        CleaningLinesSolvent1and2();

        IF bMovementComplete THEN
            eRecoveryState    := E_RecoveryState.AgitateTime2;
            iStepCounter      := 0;
            bMovementComplete := FALSE;
        END_IF


    // ----------------------------------------------------------------------
    // AgitateTime2:
    //  - Second agitation time window after lines are cleaned.
    // ----------------------------------------------------------------------
    E_RecoveryState.AgitateTime2:

        AgitateTime2();

        IF bMovementComplete THEN
            eRecoveryState    := E_RecoveryState.Prime_Needles;
            iStepCounter      := 0;
            bMovementComplete := FALSE;
        END_IF


    // ----------------------------------------------------------------------
    // Prime_Needles:
    //  - Primes the needles and final tubing before filling vials.
    // ----------------------------------------------------------------------
    E_RecoveryState.Prime_Needles:

        PrimeNeedles();

        IF bMovementComplete THEN
            eRecoveryState    := E_RecoveryState.Fill_Vials_Row_1;
            iStepCounter      := 0;
            bMovementComplete := FALSE;
        END_IF


    // ----------------------------------------------------------------------
    // Fill_Vials_Row_1:
    //  - Fills the first row of vials.
    //  - Decides next state based on how many rows must be filled
    //    (iVialsToFill from recipe).
    // ----------------------------------------------------------------------
    E_RecoveryState.Fill_Vials_Row_1:

        Fill_Vials_Row_1();

        IF bMovementComplete THEN
            IF GVL_Recipe.stCurrentRecipe.stOtherParams.iVialsToFill > 1 THEN
                eRecoveryState := E_RecoveryState.Fill_Vials_Row_2;
            ELSE
                eRecoveryState := E_RecoveryState.Waste_Remaining_Solvent;
            END_IF

            bMovementComplete := FALSE;
            iStepCounter      := 0;
        END_IF


    // ----------------------------------------------------------------------
    // Fill_Vials_Row_2:
    //  - Fills the second row of vials (if required).
    // ----------------------------------------------------------------------
    E_RecoveryState.Fill_Vials_Row_2:

        Fill_Vials_Row_2();

        IF bMovementComplete THEN
            IF GVL_Recipe.stCurrentRecipe.stOtherParams.iVialsToFill > 2 THEN
                eRecoveryState := E_RecoveryState.Fill_Vials_Row_3;
            ELSE
                eRecoveryState := E_RecoveryState.Waste_Remaining_Solvent;
            END_IF

            bMovementComplete := FALSE;
            iStepCounter      := 0;
        END_IF


    // ----------------------------------------------------------------------
    // Fill_Vials_Row_3:
    //  - Fills the third row of vials (if required).
    // ----------------------------------------------------------------------
    E_RecoveryState.Fill_Vials_Row_3:

        Fill_Vials_Row_3();

        IF bMovementComplete THEN
            IF GVL_Recipe.stCurrentRecipe.stOtherParams.iVialsToFill > 3 THEN
                eRecoveryState := E_RecoveryState.Fill_Vials_Row_4;
            ELSE
                eRecoveryState := E_RecoveryState.Waste_Remaining_Solvent;
            END_IF

            bMovementComplete := FALSE;
            iStepCounter      := 0;
        END_IF


    // ----------------------------------------------------------------------
    // Fill_Vials_Row_4:
    //  - Fills the fourth row of vials (if required).
    // ----------------------------------------------------------------------
    E_RecoveryState.Fill_Vials_Row_4:

        Fill_Vials_Row_4();

        IF bMovementComplete THEN
            eRecoveryState    := E_RecoveryState.Waste_Remaining_Solvent;
            bMovementComplete := FALSE;
            iStepCounter      := 0;
        END_IF


    // ----------------------------------------------------------------------
    // Waste_Remaining_Solvent:
    //  - Directs any remaining solvent to waste containers.
    // ----------------------------------------------------------------------
    E_RecoveryState.Waste_Remaining_Solvent:

        WasteRemainingSolvent();

        IF bMovementComplete THEN
            eRecoveryState    := E_RecoveryState.Completed;
            bMovementComplete := FALSE;
            iStepCounter      := 0;
        END_IF


    // ----------------------------------------------------------------------
    // Completed:
    //  - Recovery phase has finished successfully.
    //  - Updates HMI and raises bSuccess.
    // ----------------------------------------------------------------------
    E_RecoveryState.Completed:

        GVL_HMI.HMIAnimation.sLoadTextRecovery   := 'Completed';
        GVL_HMI.HMIAnimation.rLoadBarRecovery    := 100.0;
        GVL_HMI.HMIAnimation.eIconStateRecovery  := E_IconState.Completed;

        bSuccess := TRUE;
        // bError stays FALSE here. If you later implement error transitions
        // to a dedicated Error state, set bError accordingly there.

END_CASE

ACTION AgitateTime1:
// ==========================================================================
// AgitateTime1
// --------------------------------------------------------------------------
// Purpose:
//   - Handles the first agitation timer window for the Recovery Phase.
//   - Uses tonAgitateTime1 and sets bMovementComplete when finished.
//
// Sequence (iStepCounter):
//   0) Check if Agitate Time 1 > 0. If zero, skip directly to step 3.
//   1) Start TON timer with recipe time tAgitate1Time.
//   2) Stop TON timer and move to completion.
//   3) Raise bMovementComplete to notify the caller state.
// ==========================================================================
CASE iStepCounter OF

    0:  // Check if Agitate Time 1 is greater than zero
        IF TIME_TO_DWORD(GVL_Recipe.stActiveRecipe.stOtherParams.tAgitate1Time / 1000) > 0 THEN
            // Update HMI text
            GVL_HMI.HMIAnimation.sLoadTextRecovery := 'Agitate Time 1';
            iStepCounter := 1;
        ELSE
            // No time configured → skip timer and mark as done
            iStepCounter := 3;
        END_IF

    1:  // Start Agitate Timer 1
        tonAgitateTime1(
            IN := TRUE,
            PT := GVL_Recipe.stActiveRecipe.stOtherParams.tAgitate1Time
        );

        // When timer finishes, proceed to stop it
        IF tonAgitateTime1.Q THEN
            iStepCounter := 2;
        END_IF

    2:  // Reset Agitate Timer 1
        tonAgitateTime1(
            IN := FALSE,
            PT := GVL_Recipe.stActiveRecipe.stOtherParams.tAgitate1Time
        );
        iStepCounter := 3;

    3:  // Signal completion to Recovery FSM
        bMovementComplete := TRUE;

END_CASE
END_ACTION

ACTION AgitateTime2:
// ==========================================================================
// AgitateTime2
// --------------------------------------------------------------------------
// Purpose:
//   - Handles the second agitation timer window for the Recovery Phase.
//   - Uses tonAgitateTime2 and sets bMovementComplete when finished.
//
// Sequence (iStepCounter):
//   0) Check if Agitate Time 2 > 0. If zero, skip directly to step 3.
//   1) Start TON timer with recipe time tAgitate2Time.
//   2) Stop TON timer and move to completion.
//   3) Raise bMovementComplete to notify the caller state.
// ==========================================================================
CASE iStepCounter OF

    0:  // Check if Agitate Time 2 is greater than zero
        IF TIME_TO_DWORD(GVL_Recipe.stActiveRecipe.stOtherParams.tAgitate2Time / 1000) > 0 THEN
            // Update HMI text
            GVL_HMI.HMIAnimation.sLoadTextRecovery := 'Agitate Time 2';
            iStepCounter := 1;
        ELSE
            // No time configured → skip timer and mark as done
            iStepCounter := 3;
        END_IF

    1:  // Start Agitate Timer 2
        tonAgitateTime2(
            IN := TRUE,
            PT := GVL_Recipe.stActiveRecipe.stOtherParams.tAgitate2Time
        );

        // When timer finishes, proceed to stop it
        IF tonAgitateTime2.Q THEN
            iStepCounter := 2;
        END_IF

    2:  // Reset Agitate Timer 2
        tonAgitateTime2(
            IN := FALSE,
            PT := GVL_Recipe.stActiveRecipe.stOtherParams.tAgitate2Time
        );
        iStepCounter := 3;

    3:  // Signal completion to Recovery FSM
        bMovementComplete := TRUE;

END_CASE
END_ACTION

ACTION CleaningLinesSolvent1:
// ==========================================================================
// CleaningLinesSolvent1
// --------------------------------------------------------------------------
// Purpose:
//   - Flush / clean the fluidic lines after using Solvent 1.
//   - Moves all valves to recirculation position (5).
//   - Pumps a larger volume through all paths to clean residual solvent.
//
// Sequence (iStepCounter):
//   0) Set HMI text and prepare.
//   1) Move all valves [1..5] to position 5 (Recirculation).
//   2) Calculate pump distances based on recipe volumes (Rinse 1) + dead volume.
//   3) Run all pumps [1..10] forward with higher velocity for cleaning.
//   4) Set bMovementComplete TRUE to notify FSM.
// ==========================================================================
CASE iStepCounter OF

    0:  // Initialize action / HMI
        GVL_HMI.HMIAnimation.sLoadTextRecovery := 'Cleaning Lines R1';
        iStepCounter := 1;

    1:  // Move valves [1..5] to position 5 (Recirculation)
        FOR i := 1 TO 5 DO
            IF NOT bMoveValveDone[i] THEN
                bMoveValveDone[i] := GVL_Motion.aValvesObj[i].MoveValve(
                    iPosition := 5,
                    rVelocity := GVL_Motion.aValves[i].rTargetVel,
                    rAcc      := GVL_Motion.aValves[i].rAcceleration,
                    rDec      := GVL_Motion.aValves[i].rDeceleration
                );
            END_IF
        END_FOR

        // Wait until all valves have completed their move
        IF bMoveValveDone[1] AND bMoveValveDone[2] AND bMoveValveDone[3]
           AND bMoveValveDone[4] AND bMoveValveDone[5]
        THEN
            // Reset valve flags and move to next step
            FOR i := 1 TO 5 DO
                bMoveValveDone[i] := FALSE;
            END_FOR
            iStepCounter := 2;
        END_IF

    2:  // Calculate pump distances for cleaning (based on Rinse 1 volume)
        // Factor 1.5 is used to add margin for extra cleaning volume
		(*
        fDistance[1]  := F_VolumeToSteps((GVL_Recipe.stActiveRecipe.stVolumes.aT_IC_Volume[1] +
                                          GVL_Motion.aPumps[1].Rotary.rDeadVolume) * 1.5, 1);
										  
        fDistance[2]  := F_VolumeToSteps((GVL_Recipe.stActiveRecipe.stVolumes.aS0_Volume[1] +
                                          GVL_Motion.aPumps[2].Rotary.rDeadVolume) * 1.5, 2);
										  
        fDistance[3]  := F_VolumeToSteps((GVL_Recipe.stActiveRecipe.stVolumes.aS1_Volume[1] +
                                          GVL_Motion.aPumps[3].Rotary.rDeadVolume) * 1.5, 3);
										  
        fDistance[4]  := F_VolumeToSteps((GVL_Recipe.stActiveRecipe.stVolumes.aS2_Volume[1] +
                                          GVL_Motion.aPumps[4].Rotary.rDeadVolume) * 1.5, 4);
										  
        fDistance[5]  := F_VolumeToSteps((GVL_Recipe.stActiveRecipe.stVolumes.aS3_Volume[1] +
                                          GVL_Motion.aPumps[5].Rotary.rDeadVolume) * 1.5, 5);
										  
        fDistance[6]  := F_VolumeToSteps((GVL_Recipe.stActiveRecipe.stVolumes.aS4_Volume[1] +
                                          GVL_Motion.aPumps[6].Rotary.rDeadVolume) * 1.5, 6);
										  
        fDistance[7]  := F_VolumeToSteps((GVL_Recipe.stActiveRecipe.stVolumes.aS5_Volume[1] +
                                          GVL_Motion.aPumps[7].Rotary.rDeadVolume) * 1.5, 7);
										  
        fDistance[8]  := F_VolumeToSteps((GVL_Recipe.stActiveRecipe.stVolumes.aS6_Volume[1] +
                                          GVL_Motion.aPumps[8].Rotary.rDeadVolume) * 1.5, 8);
										  
        fDistance[9]  := F_VolumeToSteps((GVL_Recipe.stActiveRecipe.stVolumes.aS7_Volume[1] +
                                          GVL_Motion.aPumps[9].Rotary.rDeadVolume) * 1.5, 9);
										  
        fDistance[10] := F_VolumeToSteps((GVL_Recipe.stActiveRecipe.stVolumes.aF_Volume[1] +
                                          GVL_Motion.aPumps[10].Rotary.rDeadVolume) * 1.5, 10);
		*)
		
		// Constant volume for cleaning lines. change#15/01/26
		FOR i := 1 TO 10 DO
			fDistance[i]  := F_VolumeToSteps( 100 + GVL_Motion.aPumps[i].Rotary.rDeadVolume, i);
		END_FOR
		
        iStepCounter := 3;

    3:  // Start rotary pumps with calculated distances [positive movement]
        FOR i := 1 TO 10 DO
            IF NOT bMovePumpDone[i] THEN
                bMovePumpDone[i] := GVL_Motion.aPumpsRotary[i].MoveRelative(
                    Distance := fDistance[i],
                    Velocity := GVL_Settings.stPumpParameters.iRunVelocity * 6,
                    Acc      := GVL_Settings.stPumpParameters.iRunVelocity * 3,
                    Dec      := GVL_Settings.stPumpParameters.iRunVelocity * 3
                );
            END_IF
        END_FOR

        // Wait until every pump has completed the move
        IF bMovePumpDone[1] AND bMovePumpDone[2] AND bMovePumpDone[3] AND bMovePumpDone[4] AND
           bMovePumpDone[5] AND bMovePumpDone[6] AND bMovePumpDone[7] AND bMovePumpDone[8] AND
           bMovePumpDone[9] AND bMovePumpDone[10]
        THEN
            FOR i := 1 TO 10 DO
                bMovePumpDone[i] := FALSE;
            END_FOR
            iStepCounter := 4;
        END_IF

    4:  // Signal completion to Recovery FSM
        bMovementComplete := TRUE;

END_CASE
END_ACTION

ACTION CleaningLinesSolvent1and2:
// ==========================================================================
// CleaningLinesSolvent1and2
// --------------------------------------------------------------------------
// Purpose:
//   - Flush / clean all lines that carried Solvent 1 and Solvent 2.
//   - Uses the combined volumes of both rinses to determine a larger
//     cleaning volume per pump.
//
// Sequence (iStepCounter):
//   0) Set HMI text.
//   1) Move all valves [1..5] to position 5 (Recirculation).
//   2) Calculate pump distances from sum of Rinse 1 + Rinse 2 volumes.
//   3) Run all pumps [1..10] forward with higher velocity.
//   4) Set bMovementComplete TRUE.
// ==========================================================================
CASE iStepCounter OF

    0:  // Initialize action / HMI
        GVL_HMI.HMIAnimation.sLoadTextRecovery := 'Cleaning Lines';
        iStepCounter := 1;

    1:  // Move valves [1..5] to position 5 (Recirculation)
        FOR i := 1 TO 5 DO
            IF NOT bMoveValveDone[i] THEN
                bMoveValveDone[i] := GVL_Motion.aValvesObj[i].MoveValve(
                    iPosition := 5,
                    rVelocity := GVL_Motion.aValves[i].rTargetVel,
                    rAcc      := GVL_Motion.aValves[i].rAcceleration,
                    rDec      := GVL_Motion.aValves[i].rDeceleration
                );
            END_IF
        END_FOR

        IF bMoveValveDone[1] AND bMoveValveDone[2] AND bMoveValveDone[3]
           AND bMoveValveDone[4] AND bMoveValveDone[5]
        THEN
            FOR i := 1 TO 5 DO
                bMoveValveDone[i] := FALSE;
            END_FOR
            iStepCounter := 2;
        END_IF

    2:  // Calculate distances using combined volumes (Rinse 1 + Rinse 2)
        fDistance[1]  := F_VolumeToSteps((GVL_Recipe.stActiveRecipe.stVolumes.aT_IC_Volume[1] +
                                          GVL_Recipe.stActiveRecipe.stVolumes.aT_IC_Volume[2] +
                                          GVL_Motion.aPumps[1].Rotary.rDeadVolume) * 1.5, 1);
										  
        fDistance[2]  := F_VolumeToSteps((GVL_Recipe.stActiveRecipe.stVolumes.aS0_Volume[1] +
                                          GVL_Recipe.stActiveRecipe.stVolumes.aS0_Volume[2] +
                                          GVL_Motion.aPumps[2].Rotary.rDeadVolume) * 1.5, 2);
										  
        fDistance[3]  := F_VolumeToSteps((GVL_Recipe.stActiveRecipe.stVolumes.aS1_Volume[1] +
                                          GVL_Recipe.stActiveRecipe.stVolumes.aS1_Volume[2] +
                                          GVL_Motion.aPumps[3].Rotary.rDeadVolume) * 1.5, 3);
										  
        fDistance[4]  := F_VolumeToSteps((GVL_Recipe.stActiveRecipe.stVolumes.aS2_Volume[1] +
                                          GVL_Recipe.stActiveRecipe.stVolumes.aS2_Volume[2] +
                                          GVL_Motion.aPumps[4].Rotary.rDeadVolume) * 1.5, 4);
										  
        fDistance[5]  := F_VolumeToSteps((GVL_Recipe.stActiveRecipe.stVolumes.aS3_Volume[1] +
                                          GVL_Recipe.stActiveRecipe.stVolumes.aS3_Volume[2] +
                                          GVL_Motion.aPumps[5].Rotary.rDeadVolume) * 1.5, 5);
										  
        fDistance[6]  := F_VolumeToSteps((GVL_Recipe.stActiveRecipe.stVolumes.aS4_Volume[1] +
                                          GVL_Recipe.stActiveRecipe.stVolumes.aS4_Volume[2] +
                                          GVL_Motion.aPumps[6].Rotary.rDeadVolume) * 1.5, 6);
										  
        fDistance[7]  := F_VolumeToSteps((GVL_Recipe.stActiveRecipe.stVolumes.aS5_Volume[1] +
                                          GVL_Recipe.stActiveRecipe.stVolumes.aS5_Volume[2] +
                                          GVL_Motion.aPumps[7].Rotary.rDeadVolume) * 1.5, 7);
										  
        fDistance[8]  := F_VolumeToSteps((GVL_Recipe.stActiveRecipe.stVolumes.aS6_Volume[1] +
                                          GVL_Recipe.stActiveRecipe.stVolumes.aS6_Volume[2] +
                                          GVL_Motion.aPumps[8].Rotary.rDeadVolume) * 1.5, 8);
										  
        fDistance[9]  := F_VolumeToSteps((GVL_Recipe.stActiveRecipe.stVolumes.aS7_Volume[1] +
                                          GVL_Recipe.stActiveRecipe.stVolumes.aS7_Volume[2] +
                                          GVL_Motion.aPumps[9].Rotary.rDeadVolume) * 1.5, 9);
										  
        fDistance[10] := F_VolumeToSteps((GVL_Recipe.stActiveRecipe.stVolumes.aF_Volume[1] +
                                          GVL_Recipe.stActiveRecipe.stVolumes.aF_Volume[2] +
                                          GVL_Motion.aPumps[10].Rotary.rDeadVolume) * 1.5, 10);

        iStepCounter := 3;

    3:  // Run pumps with calculated distances [positive movement]
        FOR i := 1 TO 10 DO
            IF NOT bMovePumpDone[i] THEN
                bMovePumpDone[i] := GVL_Motion.aPumpsRotary[i].MoveRelative(
                    Distance := fDistance[i],
                    Velocity := GVL_Settings.stPumpParameters.iRunVelocity * 6,
                    Acc      := GVL_Settings.stPumpParameters.iRunVelocity * 3,
                    Dec      := GVL_Settings.stPumpParameters.iRunVelocity * 3
                );
            END_IF
        END_FOR

        IF bMovePumpDone[1] AND bMovePumpDone[2] AND bMovePumpDone[3] AND bMovePumpDone[4] AND
           bMovePumpDone[5] AND bMovePumpDone[6] AND bMovePumpDone[7] AND bMovePumpDone[8] AND
           bMovePumpDone[9] AND bMovePumpDone[10]
        THEN
            FOR i := 1 TO 10 DO
                bMovePumpDone[i] := FALSE;
            END_FOR
            iStepCounter := 4;
        END_IF

    4:  // Signal completion to Recovery FSM
        bMovementComplete := TRUE;

END_CASE
END_ACTION

METHOD PRIVATE EstimateTotalTime : REAL
VAR_INPUT
END_VAR
VAR
	i : INT;
	iRow : INT;
    rTotalTime : LREAL := 0.0;
    rMaxPumpTime : REAL;
    rTmpTime : REAL;
	aPumpVolume : ARRAY[1..10] OF REAL;
END_VAR
// --- MOTORS M2 and M3 ---
// Movements are sequential, so times are summed
rTotalTime := rTotalTime
    + (ABS(GVL_Settings.stMachineParam.aM2Position[3] - GVL_Settings.stMachineParam.aM2Position[1]) / GVL_Settings.stMachineParam.rM2Velocity) * 4
    + (ABS(GVL_Settings.stMachineParam.aM3Position[4] - GVL_Settings.stMachineParam.aM3Position[1]) / GVL_Settings.stMachineParam.rM3Velocity) * 4;

// --- VALVES ---
// Valves move in parallel, so estimate per group of 5 valves per switch
// Estimated 0.8s per position change, 8 total changes
rTotalTime := rTotalTime + 0.8 * 8;


// --- TIMERS ---
// Add the Agitation and Soak durations directly (in seconds)
rTotalTime := rTotalTime + TO_REAL(GVL_Recipe.stActiveRecipe.stOtherParams.tAgitate1Time) / 1000.0;
rTotalTime := rTotalTime + TO_REAL(GVL_Recipe.stActiveRecipe.stOtherParams.tAgitate2Time) / 1000.0;
rTotalTime := rTotalTime + TO_REAL(GVL_Recipe.stActiveRecipe.stOtherParams.tSoakTime) / 1000.0;


// --- PUMPS ---
// Pumps move in parallel. We always use the slowest pump as reference for each phase.

// Metering Solvent 1
rMaxPumpTime := 0;
aPumpVolume[1] := GVL_Recipe.stActiveRecipe.stVolumes.aT_IC_Volume[1] + 10;
aPumpVolume[2] := GVL_Recipe.stActiveRecipe.stVolumes.aS0_Volume[1] + 10;
aPumpVolume[3] := GVL_Recipe.stActiveRecipe.stVolumes.aS1_Volume[1] + 10;
aPumpVolume[4] := GVL_Recipe.stActiveRecipe.stVolumes.aS2_Volume[1] + 10;
aPumpVolume[5] := GVL_Recipe.stActiveRecipe.stVolumes.aS3_Volume[1] + 10;
aPumpVolume[6] := GVL_Recipe.stActiveRecipe.stVolumes.aS4_Volume[1] + 10;
aPumpVolume[7] := GVL_Recipe.stActiveRecipe.stVolumes.aS5_Volume[1] + 10;
aPumpVolume[8] := GVL_Recipe.stActiveRecipe.stVolumes.aS6_Volume[1] + 10;
aPumpVolume[9] := GVL_Recipe.stActiveRecipe.stVolumes.aS7_Volume[1] + 10;
aPumpVolume[10] := GVL_Recipe.stActiveRecipe.stVolumes.aF_Volume[1] + 10;

FOR i := 1 TO 10 DO
    rTmpTime := F_VolumeToSteps(rVolume := aPumpVolume[i], iPumpIndex := i) / GVL_Motion.aPumps[i].Rotary.rSpeed;
    IF rTmpTime > rMaxPumpTime THEN rMaxPumpTime := rTmpTime; END_IF
END_FOR
rTotalTime := rTotalTime + rMaxPumpTime;

// Metering Solvent 2
rMaxPumpTime := 0;
aPumpVolume[1] := GVL_Recipe.stActiveRecipe.stVolumes.aT_IC_Volume[2] + 10;
aPumpVolume[2] := GVL_Recipe.stActiveRecipe.stVolumes.aS0_Volume[2] + 10;
aPumpVolume[3] := GVL_Recipe.stActiveRecipe.stVolumes.aS1_Volume[2] + 10;
aPumpVolume[4] := GVL_Recipe.stActiveRecipe.stVolumes.aS2_Volume[2] + 10;
aPumpVolume[5] := GVL_Recipe.stActiveRecipe.stVolumes.aS3_Volume[2] + 10;
aPumpVolume[6] := GVL_Recipe.stActiveRecipe.stVolumes.aS4_Volume[2] + 10;
aPumpVolume[7] := GVL_Recipe.stActiveRecipe.stVolumes.aS5_Volume[2] + 10;
aPumpVolume[8] := GVL_Recipe.stActiveRecipe.stVolumes.aS6_Volume[2] + 10;
aPumpVolume[9] := GVL_Recipe.stActiveRecipe.stVolumes.aS7_Volume[2] + 10;
aPumpVolume[10] := GVL_Recipe.stActiveRecipe.stVolumes.aF_Volume[2] + 10;
FOR i := 1 TO 10 DO
    rTmpTime := F_VolumeToSteps(rVolume := aPumpVolume[i], iPumpIndex := i) / GVL_Motion.aPumps[i].Rotary.rSpeed;
    IF rTmpTime > rMaxPumpTime THEN rMaxPumpTime := rTmpTime; END_IF
END_FOR
rTotalTime := rTotalTime + rMaxPumpTime;

// Prime Needles
rMaxPumpTime := 0;
FOR i := 1 TO 10 DO
    rTmpTime := F_VolumeToSteps(rVolume := GVL_Recipe.stActiveRecipe.stOtherParams.rVialPrimeVol + 20, iPumpIndex := i) / GVL_Motion.aPumps[i].Rotary.rSpeed;
    IF rTmpTime > rMaxPumpTime THEN rMaxPumpTime := rTmpTime; END_IF
END_FOR
rTotalTime := rTotalTime + rMaxPumpTime;

// Fill Vials Rows 1–4
FOR iRow := 1 TO GVL_Recipe.stActiveRecipe.stOtherParams.iVialsToFill DO
    rMaxPumpTime := 0;
    FOR i := 1 TO 10 DO
        IF iRow = 1 THEN
            rTmpTime := F_VolumeToSteps(rVolume := GVL_Recipe.stActiveRecipe.stOtherParams.rVial1FillVol, iPumpIndex := i) / GVL_Motion.aPumps[i].Rotary.rSpeed;
        ELSE
            rTmpTime := F_VolumeToSteps(rVolume := GVL_Recipe.stActiveRecipe.stOtherParams.rVials2_4FillVol, iPumpIndex := i) / GVL_Motion.aPumps[i].Rotary.rSpeed;
        END_IF
        IF rTmpTime > rMaxPumpTime THEN 
			rMaxPumpTime := rTmpTime; 
		END_IF
    END_FOR
    rTotalTime := rTotalTime + rMaxPumpTime;
END_FOR

// Waste Remaining Solvent
rMaxPumpTime := 0;

FOR i := 1 TO 10 DO
    rTmpTime := F_VolumeToSteps(rVolume := GVL_Recipe.stActiveRecipe.stVolumes.aT_IC_Volume[1] + GVL_Recipe.stActiveRecipe.stVolumes.aT_IC_Volume[2], iPumpIndex := i) / GVL_Motion.aPumps[i].Rotary.rSpeed;
    IF rTmpTime > rMaxPumpTime THEN
 		rMaxPumpTime := rTmpTime; 
	END_IF
	
END_FOR
rTotalTime := rTotalTime + rMaxPumpTime;

EstimateTotalTime := rTotalTime + 180;
END_METHOD

ACTION Fill_Vials_Row_1:
// ==========================================================================
// Fill_Vials_Row_1
// --------------------------------------------------------------------------
// Purpose:
//   - Fill the first row of vials using the Recovery Phase solvent mixture.
//   - Move M3 (horizontal) to vial row 1 position and M2 (vertical) down to
//     the vial level.
//   - Pump the volume configured as rVial1FillVol into each vial.
//
// Sequence (iStepCounter):
//   0) Initialize HMI text and move to step 1.
//   1) Set all valves [1..5] to position 6 (Needles).
//   2) Move M3 to vial row 1 (horizontal) and M2 down to vial height.
//   3) Compute pump distances based on rVial1FillVol.
//   4) Run pumps [1..10] backward (negative Distance) to dispense volume.
//   5) Move M2 back to home (vertical).
//   6) Set bMovementComplete := TRUE to notify the Recovery FSM.
// ==========================================================================
CASE iStepCounter OF

    0: // Initialize HMI info for Row 1 filling
        GVL_HMI.HMIAnimation.sLoadTextRecovery := 'Fill Vials R1';
        // Optionally: GVL_HMI.HMIAnimation.rLoadBarRecovery := 70;
        iStepCounter := 1;

    1: // Set valves [1..5] to position 6 (Needles)
        FOR i := 1 TO 5 DO
            IF NOT bMoveValveDone[i] THEN
                bMoveValveDone[i] := GVL_Motion.aValvesObj[i].MoveValve(
                    iPosition := 6,
                    rVelocity := GVL_Motion.aValves[i].rTargetVel,
                    rAcc      := GVL_Motion.aValves[i].rAcceleration,
                    rDec      := GVL_Motion.aValves[i].rDeceleration
                );
            END_IF
        END_FOR

        // Wait for all valves to finish the movement
        IF bMoveValveDone[1] AND bMoveValveDone[2] AND bMoveValveDone[3]
           AND bMoveValveDone[4] AND bMoveValveDone[5]
        THEN
            // Reset valve flags and go to next step
            FOR i := 1 TO 5 DO
                bMoveValveDone[i] := FALSE;
            END_FOR
            iStepCounter := 2;
        END_IF

    2: // M2 and M3 motors movement to vial row 1 position
        // Step 2.1: Move M3 (horizontal) to Row 1 (AboveVialSet1)
        IF NOT bMoveM3 THEN
            bMoveM3 := GVL_Motion.aMotors[3].MoveAbsolute(
                rPosition := GVL_Settings.stMachineParam.aM3Position[2], // Vial row 1
                rVelocity := GVL_Settings.stMachineParam.rM3Velocity,
                rAcc      := GVL_Settings.stMachineParam.rM3Accleration,
                rDec      := GVL_Settings.stMachineParam.rM3Deceleration
            );
        END_IF

        // Step 2.2: After M3 is at row 1, move M2 (vertical) down to vial height
        IF NOT bMoveM2 AND bMoveM3 THEN
            bMoveM2 := GVL_Motion.aMotors[2].MoveAbsolute(
                rPosition := GVL_Settings.stMachineParam.aM2Position[3], // Fill position
                rVelocity := GVL_Settings.stMachineParam.rM2Velocity,
                rAcc      := GVL_Settings.stMachineParam.rM2Accleration,
                rDec      := GVL_Settings.stMachineParam.rM2Deceleration
            );
        END_IF

        // When both motors reach their positions, clear flags and go to step 3
        IF bMoveM2 AND bMoveM3 THEN
            bMoveM2      := FALSE;
            bMoveM3      := FALSE;
            iStepCounter := 3;
        END_IF

    3: // Calculate distance (steps) for each pump based on rVial1FillVol
        fDistance[1]  := F_VolumeToSteps(
            rVolume    := GVL_Recipe.stActiveRecipe.stOtherParams.rVial1FillVol,
            iPumpIndex := 1
        );
        fDistance[2]  := F_VolumeToSteps(
            rVolume    := GVL_Recipe.stActiveRecipe.stOtherParams.rVial1FillVol,
            iPumpIndex := 2
        );
        fDistance[3]  := F_VolumeToSteps(
            rVolume    := GVL_Recipe.stActiveRecipe.stOtherParams.rVial1FillVol,
            iPumpIndex := 3
        );
        fDistance[4]  := F_VolumeToSteps(
            rVolume    := GVL_Recipe.stActiveRecipe.stOtherParams.rVial1FillVol,
            iPumpIndex := 4
        );
        fDistance[5]  := F_VolumeToSteps(
            rVolume    := GVL_Recipe.stActiveRecipe.stOtherParams.rVial1FillVol,
            iPumpIndex := 5
        );
        fDistance[6]  := F_VolumeToSteps(
            rVolume    := GVL_Recipe.stActiveRecipe.stOtherParams.rVial1FillVol,
            iPumpIndex := 6
        );
        fDistance[7]  := F_VolumeToSteps(
            rVolume    := GVL_Recipe.stActiveRecipe.stOtherParams.rVial1FillVol,
            iPumpIndex := 7
        );
        fDistance[8]  := F_VolumeToSteps(
            rVolume    := GVL_Recipe.stActiveRecipe.stOtherParams.rVial1FillVol,
            iPumpIndex := 8
        );
        fDistance[9]  := F_VolumeToSteps(
            rVolume    := GVL_Recipe.stActiveRecipe.stOtherParams.rVial1FillVol,
            iPumpIndex := 9
        );
        fDistance[10] := F_VolumeToSteps(
            rVolume    := GVL_Recipe.stActiveRecipe.stOtherParams.rVial1FillVol,
            iPumpIndex := 10
        );

        iStepCounter := 4;

    4: // Pump by distance (deg/s → steps) [negative movement = dispensing to vials]
        FOR i := 1 TO 10 DO
            IF NOT bMovePumpDone[i] THEN
                bMovePumpDone[i] := GVL_Motion.aPumpsRotary[i].MoveRelative(
                    Distance := -fDistance[i],   // negative → pushing out to vials
                    Velocity := GVL_Settings.stPumpParameters.iMeterVelocity * 6,
                    Acc      := GVL_Settings.stPumpParameters.iMeterVelocity * 3,
                    Dec      := GVL_Settings.stPumpParameters.iMeterVelocity * 3
                );
            END_IF
        END_FOR

        // Wait until all pumps finish their moves
        IF bMovePumpDone[1]  AND bMovePumpDone[2]  AND bMovePumpDone[3]  AND
           bMovePumpDone[4]  AND bMovePumpDone[5]  AND bMovePumpDone[6]  AND
           bMovePumpDone[7]  AND bMovePumpDone[8]  AND bMovePumpDone[9]  AND
           bMovePumpDone[10]
        THEN
            FOR i := 1 TO 10 DO
                bMovePumpDone[i] := FALSE;
            END_FOR
            iStepCounter := 5;
        END_IF

    5: // Move M2 (vertical) back to home position
        IF NOT bMoveM2 THEN
            bMoveM2 := GVL_Motion.aMotors[2].MoveAbsolute(
                rPosition := GVL_Settings.stMachineParam.aM2Position[1], // home
                rVelocity := GVL_Settings.stMachineParam.rM2Velocity,
                rAcc      := GVL_Settings.stMachineParam.rM2Accleration,
                rDec      := GVL_Settings.stMachineParam.rM2Deceleration
            );
        END_IF

        // When M2 is home, clear flag and go to final step
        IF bMoveM2 THEN
            bMoveM2      := FALSE;
            iStepCounter := 6;
        END_IF

    6: // Notify Recovery FSM that Row 1 filling is completed
        bMovementComplete := TRUE;

END_CASE
END_ACTION

ACTION Fill_Vials_Row_2:
// ==========================================================================
// Fill_Vials_Row_2
// --------------------------------------------------------------------------
// Purpose:
//   - Fill the second row of vials using the same volume used for rows 2–4.
//   - Move M3 (horizontal) to vial row 2 and M2 (vertical) down to vial level.
//   - Pump the volume configured as rVials2_4FillVol into each vial.
//
// Sequence (iStepCounter):
//   0) Initialize HMI text and move to step 1.
//   1) Set all valves [1..5] to position 6 (Needles).
//   2) Move M3 to vial row 2 (AboveVialSet1 + VialSetSpacing) and M2 down.
//   3) Compute pump distances based on rVials2_4FillVol.
//   4) Run pumps [1..10] backward to dispense volume.
//   5) Move M2 back to home (vertical).
//   6) Set bMovementComplete := TRUE.
// ==========================================================================
CASE iStepCounter OF

    0: // Initialize HMI info for Row 2 filling
        GVL_HMI.HMIAnimation.sLoadTextRecovery := 'Fill Vials R2';
        // Optionally: GVL_HMI.HMIAnimation.rLoadBarRecovery := 75;
        iStepCounter := 1;

    1: // Set valves [1..5] to position 6 (Needles)
        FOR i := 1 TO 5 DO
            IF NOT bMoveValveDone[i] THEN
                bMoveValveDone[i] := GVL_Motion.aValvesObj[i].MoveValve(
                    iPosition := 6,
                    rVelocity := GVL_Motion.aValves[i].rTargetVel,
                    rAcc      := GVL_Motion.aValves[i].rAcceleration,
                    rDec      := GVL_Motion.aValves[i].rDeceleration
                );
            END_IF
        END_FOR

        IF bMoveValveDone[1] AND bMoveValveDone[2] AND bMoveValveDone[3]
           AND bMoveValveDone[4] AND bMoveValveDone[5]
        THEN
            FOR i := 1 TO 5 DO
                bMoveValveDone[i] := FALSE;
            END_FOR
            iStepCounter := 2;
        END_IF

    2: // M2 and M3 movement to vial row 2
        // Step 2.1: M3 → row 2 = AboveVialSet1 + 1 * VialSetSpacing
        IF NOT bMoveM3 THEN
            bMoveM3 := GVL_Motion.aMotors[3].MoveAbsolute(
                rPosition := GVL_Settings.stMachineParam.aM3Position[2] +
                             (1 * GVL_Settings.stMachineParam.aM3Position[3]),
                // comment: AboveVialSet1 + (1 * VialSetSpacing)
                rVelocity := GVL_Settings.stMachineParam.rM3Velocity,
                rAcc      := GVL_Settings.stMachineParam.rM3Accleration,
                rDec      := GVL_Settings.stMachineParam.rM3Deceleration
            );
        END_IF

        // Step 2.2: after M3 movement, bring M2 down to fill position
        IF NOT bMoveM2 AND bMoveM3 THEN
            bMoveM2 := GVL_Motion.aMotors[2].MoveAbsolute(
                rPosition := GVL_Settings.stMachineParam.aM2Position[3], // Fill position
                rVelocity := GVL_Settings.stMachineParam.rM2Velocity,
                rAcc      := GVL_Settings.stMachineParam.rM2Accleration,
                rDec      := GVL_Settings.stMachineParam.rM2Deceleration
            );
        END_IF

        IF bMoveM2 AND bMoveM3 THEN
            bMoveM2      := FALSE;
            bMoveM3      := FALSE;
            iStepCounter := 3;
        END_IF

    3: // Calculate distances for each pump based on rVials2_4FillVol
        fDistance[1]  := F_VolumeToSteps(
            rVolume    := GVL_Recipe.stActiveRecipe.stOtherParams.rVials2_4FillVol,
            iPumpIndex := 1
        );
        fDistance[2]  := F_VolumeToSteps(
            rVolume    := GVL_Recipe.stActiveRecipe.stOtherParams.rVials2_4FillVol,
            iPumpIndex := 2
        );
        fDistance[3]  := F_VolumeToSteps(
            rVolume    := GVL_Recipe.stActiveRecipe.stOtherParams.rVials2_4FillVol,
            iPumpIndex := 3
        );
        fDistance[4]  := F_VolumeToSteps(
            rVolume    := GVL_Recipe.stActiveRecipe.stOtherParams.rVials2_4FillVol,
            iPumpIndex := 4
        );
        fDistance[5]  := F_VolumeToSteps(
            rVolume    := GVL_Recipe.stActiveRecipe.stOtherParams.rVials2_4FillVol,
            iPumpIndex := 5
        );
        fDistance[6]  := F_VolumeToSteps(
            rVolume    := GVL_Recipe.stActiveRecipe.stOtherParams.rVials2_4FillVol,
            iPumpIndex := 6
        );
        fDistance[7]  := F_VolumeToSteps(
            rVolume    := GVL_Recipe.stActiveRecipe.stOtherParams.rVials2_4FillVol,
            iPumpIndex := 7
        );
        fDistance[8]  := F_VolumeToSteps(
            rVolume    := GVL_Recipe.stActiveRecipe.stOtherParams.rVials2_4FillVol,
            iPumpIndex := 8
        );
        fDistance[9]  := F_VolumeToSteps(
            rVolume    := GVL_Recipe.stActiveRecipe.stOtherParams.rVials2_4FillVol,
            iPumpIndex := 9
        );
        fDistance[10] := F_VolumeToSteps(
            rVolume    := GVL_Recipe.stActiveRecipe.stOtherParams.rVials2_4FillVol,
            iPumpIndex := 10
        );

        iStepCounter := 4;

    4: // Pump by distance (negative movement = dispensing to vials)
        FOR i := 1 TO 10 DO
            IF NOT bMovePumpDone[i] THEN
                bMovePumpDone[i] := GVL_Motion.aPumpsRotary[i].MoveRelative(
                    Distance := -fDistance[i],
                    Velocity := GVL_Settings.stPumpParameters.iMeterVelocity * 6,
                    Acc      := GVL_Settings.stPumpParameters.iMeterVelocity * 3,
                    Dec      := GVL_Settings.stPumpParameters.iMeterVelocity * 3
                );
            END_IF
        END_FOR

        IF bMovePumpDone[1]  AND bMovePumpDone[2]  AND bMovePumpDone[3]  AND
           bMovePumpDone[4]  AND bMovePumpDone[5]  AND bMovePumpDone[6]  AND
           bMovePumpDone[7]  AND bMovePumpDone[8]  AND bMovePumpDone[9]  AND
           bMovePumpDone[10]
        THEN
            FOR i := 1 TO 10 DO
                bMovePumpDone[i] := FALSE;
            END_FOR
            iStepCounter := 5;
        END_IF

    5: // Move M2 back to home position
        IF NOT bMoveM2 THEN
            bMoveM2 := GVL_Motion.aMotors[2].MoveAbsolute(
                rPosition := GVL_Settings.stMachineParam.aM2Position[1], // home
                rVelocity := GVL_Settings.stMachineParam.rM2Velocity,
                rAcc      := GVL_Settings.stMachineParam.rM2Accleration,
                rDec      := GVL_Settings.stMachineParam.rM2Deceleration
            );
        END_IF

        IF bMoveM2 THEN
            bMoveM2      := FALSE;
            iStepCounter := 6;
        END_IF

    6: // Notify Recovery FSM that Row 2 filling is completed
        bMovementComplete := TRUE;

END_CASE
END_ACTION

ACTION Fill_Vials_Row_3:
// ==========================================================================
// Fill_Vials_Row_3
// --------------------------------------------------------------------------
// Purpose:
//   - Fill the third row of vials using rVials2_4FillVol.
//   - Move M3 (horizontal) to row 3 and M2 (vertical) down to vials.
//   - Pump the configured volume into each vial.
//
// Sequence (iStepCounter):
//   0) Initialize HMI text.
//   1) Set valves [1..5] to position 6 (Needles).
//   2) Move M3 to vial row 3 (AboveVialSet1 + 2 * VialSetSpacing) and M2 down.
//   3) Compute pump distances based on rVials2_4FillVol.
//   4) Pump backward to dispense.
//   5) Move M2 back to home.
//   6) bMovementComplete := TRUE.
// ==========================================================================
CASE iStepCounter OF

    0: // Initialize HMI info for Row 3 filling
        GVL_HMI.HMIAnimation.sLoadTextRecovery := 'Fill Vials R3';
        iStepCounter := 1;

    1: // Set valves [1..5] to position 6 (Needles)
        FOR i := 1 TO 5 DO
            IF NOT bMoveValveDone[i] THEN
                bMoveValveDone[i] := GVL_Motion.aValvesObj[i].MoveValve(
                    iPosition := 6,
                    rVelocity := GVL_Motion.aValves[i].rTargetVel,
                    rAcc      := GVL_Motion.aValves[i].rAcceleration,
                    rDec      := GVL_Motion.aValves[i].rDeceleration
                );
            END_IF
        END_FOR

        IF bMoveValveDone[1] AND bMoveValveDone[2] AND bMoveValveDone[3]
           AND bMoveValveDone[4] AND bMoveValveDone[5]
        THEN
            FOR i := 1 TO 5 DO
                bMoveValveDone[i] := FALSE;
            END_FOR
            iStepCounter := 2;
        END_IF

    2: // M2 and M3 movement to vial row 3
        // Step 2.1: M3 → row 3 = AboveVialSet1 + 2 * VialSetSpacing
        IF NOT bMoveM3 THEN
            bMoveM3 := GVL_Motion.aMotors[3].MoveAbsolute(
                rPosition := GVL_Settings.stMachineParam.aM3Position[2] +
                             (2 * GVL_Settings.stMachineParam.aM3Position[3]),
                // comment: AboveVialSet1 + (2 * VialSetSpacing)
                rVelocity := GVL_Settings.stMachineParam.rM3Velocity,
                rAcc      := GVL_Settings.stMachineParam.rM3Accleration,
                rDec      := GVL_Settings.stMachineParam.rM3Deceleration
            );
        END_IF

        // Step 2.2: after M3 movement, bring M2 down to fill position
        IF NOT bMoveM2 AND bMoveM3 THEN
            bMoveM2 := GVL_Motion.aMotors[2].MoveAbsolute(
                rPosition := GVL_Settings.stMachineParam.aM2Position[3], // Fill position
                rVelocity := GVL_Settings.stMachineParam.rM2Velocity,
                rAcc      := GVL_Settings.stMachineParam.rM2Accleration,
                rDec      := GVL_Settings.stMachineParam.rM2Deceleration
            );
        END_IF

        IF bMoveM2 AND bMoveM3 THEN
            bMoveM2      := FALSE;
            bMoveM3      := FALSE;
            iStepCounter := 3;
        END_IF

    3: // Calculate distances for each pump based on rVials2_4FillVol
        fDistance[1]  := F_VolumeToSteps(
            rVolume    := GVL_Recipe.stActiveRecipe.stOtherParams.rVials2_4FillVol,
            iPumpIndex := 1
        );
        fDistance[2]  := F_VolumeToSteps(
            rVolume    := GVL_Recipe.stActiveRecipe.stOtherParams.rVials2_4FillVol,
            iPumpIndex := 2
        );
        fDistance[3]  := F_VolumeToSteps(
            rVolume    := GVL_Recipe.stActiveRecipe.stOtherParams.rVials2_4FillVol,
            iPumpIndex := 3
        );
        fDistance[4]  := F_VolumeToSteps(
            rVolume    := GVL_Recipe.stActiveRecipe.stOtherParams.rVials2_4FillVol,
            iPumpIndex := 4
        );
        fDistance[5]  := F_VolumeToSteps(
            rVolume    := GVL_Recipe.stActiveRecipe.stOtherParams.rVials2_4FillVol,
            iPumpIndex := 5
        );
        fDistance[6]  := F_VolumeToSteps(
            rVolume    := GVL_Recipe.stActiveRecipe.stOtherParams.rVials2_4FillVol,
            iPumpIndex := 6
        );
        fDistance[7]  := F_VolumeToSteps(
            rVolume    := GVL_Recipe.stActiveRecipe.stOtherParams.rVials2_4FillVol,
            iPumpIndex := 7
        );
        fDistance[8]  := F_VolumeToSteps(
            rVolume    := GVL_Recipe.stActiveRecipe.stOtherParams.rVials2_4FillVol,
            iPumpIndex := 8
        );
        fDistance[9]  := F_VolumeToSteps(
            rVolume    := GVL_Recipe.stActiveRecipe.stOtherParams.rVials2_4FillVol,
            iPumpIndex := 9
        );
        fDistance[10] := F_VolumeToSteps(
            rVolume    := GVL_Recipe.stActiveRecipe.stOtherParams.rVials2_4FillVol,
            iPumpIndex := 10
        );

        iStepCounter := 4;

    4: // Pump by distance (negative movement = dispensing to vials)
        FOR i := 1 TO 10 DO
            IF NOT bMovePumpDone[i] THEN
                bMovePumpDone[i] := GVL_Motion.aPumpsRotary[i].MoveRelative(
                    Distance := -fDistance[i],
                    Velocity := GVL_Settings.stPumpParameters.iMeterVelocity * 6,
                    Acc      := GVL_Settings.stPumpParameters.iMeterVelocity * 3,
                    Dec      := GVL_Settings.stPumpParameters.iMeterVelocity * 3
                );
            END_IF
        END_FOR

        IF bMovePumpDone[1]  AND bMovePumpDone[2]  AND bMovePumpDone[3]  AND
           bMovePumpDone[4]  AND bMovePumpDone[5]  AND bMovePumpDone[6]  AND
           bMovePumpDone[7]  AND bMovePumpDone[8]  AND bMovePumpDone[9]  AND
           bMovePumpDone[10]
        THEN
            FOR i := 1 TO 10 DO
                bMovePumpDone[i] := FALSE;
            END_FOR
            iStepCounter := 5;
        END_IF

    5: // Move M2 back to home position
        IF NOT bMoveM2 THEN
            bMoveM2 := GVL_Motion.aMotors[2].MoveAbsolute(
                rPosition := GVL_Settings.stMachineParam.aM2Position[1],
                rVelocity := GVL_Settings.stMachineParam.rM2Velocity,
                rAcc      := GVL_Settings.stMachineParam.rM2Accleration,
                rDec      := GVL_Settings.stMachineParam.rM2Deceleration
            );
        END_IF

        IF bMoveM2 THEN
            bMoveM2      := FALSE;
            iStepCounter := 6;
        END_IF

    6: // Notify Recovery FSM that Row 3 filling is completed
        bMovementComplete := TRUE;

END_CASE
END_ACTION

ACTION Fill_Vials_Row_4:
// ==========================================================================
// Fill_Vials_Row_4
// --------------------------------------------------------------------------
// Purpose:
//   - Fill the fourth row of vials using rVials2_4FillVol.
//   - Move M3 (horizontal) to row 4 and M2 (vertical) down to vials.
//   - Pump the configured volume into each vial.
//
// Sequence (iStepCounter):
//   0) Initialize HMI text.
//   1) Set valves [1..5] to position 6 (Needles).
//   2) Move M3 to vial row 4 (AboveVialSet1 + 3 * VialSetSpacing) and M2 down.
//   3) Compute pump distances based on rVials2_4FillVol.
//   4) Pump backward to dispense.
//   5) Move M2 back to home.
//   6) bMovementComplete := TRUE.
// ==========================================================================
CASE iStepCounter OF

    0: // Initialize HMI info for Row 4 filling
        GVL_HMI.HMIAnimation.sLoadTextRecovery := 'Fill Vials R4';
        iStepCounter := 1;

    1: // Set valves [1..5] to position 6 (Needles)
        FOR i := 1 TO 5 DO
            IF NOT bMoveValveDone[i] THEN
                bMoveValveDone[i] := GVL_Motion.aValvesObj[i].MoveValve(
                    iPosition := 6,
                    rVelocity := GVL_Motion.aValves[i].rTargetVel,
                    rAcc      := GVL_Motion.aValves[i].rAcceleration,
                    rDec      := GVL_Motion.aValves[i].rDeceleration
                );
            END_IF
        END_FOR

        IF bMoveValveDone[1] AND bMoveValveDone[2] AND bMoveValveDone[3]
           AND bMoveValveDone[4] AND bMoveValveDone[5]
        THEN
            FOR i := 1 TO 5 DO
                bMoveValveDone[i] := FALSE;
            END_FOR
            iStepCounter := 2;
        END_IF

    2: // M2 and M3 movement to vial row 4
        // Step 2.1: M3 → row 4 = AboveVialSet1 + 3 * VialSetSpacing
        IF NOT bMoveM3 THEN
            bMoveM3 := GVL_Motion.aMotors[3].MoveAbsolute(
                rPosition := GVL_Settings.stMachineParam.aM3Position[2] +
                             (3 * GVL_Settings.stMachineParam.aM3Position[3]),
                // comment: AboveVialSet1 + (3 * VialSetSpacing)
                rVelocity := GVL_Settings.stMachineParam.rM3Velocity,
                rAcc      := GVL_Settings.stMachineParam.rM3Accleration,
                rDec      := GVL_Settings.stMachineParam.rM3Deceleration
            );
        END_IF

        // Step 2.2: M2 down to fill position after M3 movement
        IF NOT bMoveM2 AND bMoveM3 THEN
            bMoveM2 := GVL_Motion.aMotors[2].MoveAbsolute(
                rPosition := GVL_Settings.stMachineParam.aM2Position[3], // Fill position
                rVelocity := GVL_Settings.stMachineParam.rM2Velocity,
                rAcc      := GVL_Settings.stMachineParam.rM2Accleration,
                rDec      := GVL_Settings.stMachineParam.rM2Deceleration
            );
        END_IF

        IF bMoveM2 AND bMoveM3 THEN
            bMoveM2      := FALSE;
            bMoveM3      := FALSE;
            iStepCounter := 3;
        END_IF

    3: // Calculate distances for each pump based on rVials2_4FillVol
        fDistance[1]  := F_VolumeToSteps(
            rVolume    := GVL_Recipe.stActiveRecipe.stOtherParams.rVials2_4FillVol,
            iPumpIndex := 1
        );
        fDistance[2]  := F_VolumeToSteps(
            rVolume    := GVL_Recipe.stActiveRecipe.stOtherParams.rVials2_4FillVol,
            iPumpIndex := 2
        );
        fDistance[3]  := F_VolumeToSteps(
            rVolume    := GVL_Recipe.stActiveRecipe.stOtherParams.rVials2_4FillVol,
            iPumpIndex := 3
        );
        fDistance[4]  := F_VolumeToSteps(
            rVolume    := GVL_Recipe.stActiveRecipe.stOtherParams.rVials2_4FillVol,
            iPumpIndex := 4
        );
        fDistance[5]  := F_VolumeToSteps(
            rVolume    := GVL_Recipe.stActiveRecipe.stOtherParams.rVials2_4FillVol,
            iPumpIndex := 5
        );
        fDistance[6]  := F_VolumeToSteps(
            rVolume    := GVL_Recipe.stActiveRecipe.stOtherParams.rVials2_4FillVol,
            iPumpIndex := 6
        );
        fDistance[7]  := F_VolumeToSteps(
            rVolume    := GVL_Recipe.stActiveRecipe.stOtherParams.rVials2_4FillVol,
            iPumpIndex := 7
        );
        fDistance[8]  := F_VolumeToSteps(
            rVolume    := GVL_Recipe.stActiveRecipe.stOtherParams.rVials2_4FillVol,
            iPumpIndex := 8
        );
        fDistance[9]  := F_VolumeToSteps(
            rVolume    := GVL_Recipe.stActiveRecipe.stOtherParams.rVials2_4FillVol,
            iPumpIndex := 9
        );
        fDistance[10] := F_VolumeToSteps(
            rVolume    := GVL_Recipe.stActiveRecipe.stOtherParams.rVials2_4FillVol,
            iPumpIndex := 10
        );

        iStepCounter := 4;

    4: // Pump by distance (negative movement = dispensing to vials)
        FOR i := 1 TO 10 DO
            IF NOT bMovePumpDone[i] THEN
                bMovePumpDone[i] := GVL_Motion.aPumpsRotary[i].MoveRelative(
                    Distance := -fDistance[i],
                    Velocity := GVL_Settings.stPumpParameters.iMeterVelocity * 6,
                    Acc      := GVL_Settings.stPumpParameters.iMeterVelocity * 3,
                    Dec      := GVL_Settings.stPumpParameters.iMeterVelocity * 3
                );
            END_IF
        END_FOR

        IF bMovePumpDone[1]  AND bMovePumpDone[2]  AND bMovePumpDone[3]  AND
           bMovePumpDone[4]  AND bMovePumpDone[5]  AND bMovePumpDone[6]  AND
           bMovePumpDone[7]  AND bMovePumpDone[8]  AND bMovePumpDone[9]  AND
           bMovePumpDone[10]
        THEN
            FOR i := 1 TO 10 DO
                bMovePumpDone[i] := FALSE;
            END_FOR
            iStepCounter := 5;
        END_IF

    5: // Move M2 back to home position
        IF NOT bMoveM2 THEN
            bMoveM2 := GVL_Motion.aMotors[2].MoveAbsolute(
                rPosition := GVL_Settings.stMachineParam.aM2Position[1],
                rVelocity := GVL_Settings.stMachineParam.rM2Velocity,
                rAcc      := GVL_Settings.stMachineParam.rM2Accleration,
                rDec      := GVL_Settings.stMachineParam.rM2Deceleration
            );
        END_IF

        IF bMoveM2 THEN
            bMoveM2      := FALSE;
            iStepCounter := 6;
        END_IF

    6: // Notify Recovery FSM that Row 4 filling is completed
        bMovementComplete := TRUE;

END_CASE
END_ACTION

METHOD PRIVATE GetPumpVolume : REAL
VAR_INPUT
	iPump : INT;  // Pump number 1..10
    iStep : INT;  // 1..4 [step Rinse 1 | Rinse 2 | Wash 1 | Wash 2] 
END_VAR
VAR
    volume : REAL;
END_VAR
CASE iPump OF
    1: volume := GVL_Recipe.stVolumes.aT_IC_Volume[iStep];
    2: volume := GVL_Recipe.stVolumes.aS0_Volume[iStep];
    3: volume := GVL_Recipe.stVolumes.aS1_Volume[iStep];
    4: volume := GVL_Recipe.stVolumes.aS2_Volume[iStep];
    5: volume := GVL_Recipe.stVolumes.aS3_Volume[iStep];
    6: volume := GVL_Recipe.stVolumes.aS4_Volume[iStep];
    7: volume := GVL_Recipe.stVolumes.aS5_Volume[iStep];
    8: volume := GVL_Recipe.stVolumes.aS6_Volume[iStep];
    9: volume := GVL_Recipe.stVolumes.aS7_Volume[iStep];
    10: volume := GVL_Recipe.stVolumes.aF_Volume[iStep];
    ELSE
        volume := 0.0;
END_CASE

GetPumpVolume := volume;
END_METHOD

ACTION MeteringSolvent1:
// ==========================================================================
// MeteringSolvent1
// --------------------------------------------------------------------------
// Purpose:
//   - Meter Solvent 1 volumes from each Andersen stage into the fluidic path.
//   - Positions valves according to recipe aSolventN[1].
//   - Moves all 10 pumps by a distance equivalent to the configured volumes.
//
// Sequence (iStepCounter):
//   0) Set HMI text.
//   1) Ensure solenoids are in IDLE position (via gSetSolenoidControl.Idle()).
//   2) Move all valves [1..5] to solvent-1 position (recipe-dependent).
//   3) Calculate pump distances for metering (Rinse 1 + dead volume).
//   4) Run all pumps forward at metering velocity.
//   5) Set bMovementComplete TRUE.
// ==========================================================================
CASE iStepCounter OF

    0:  // Initialize action / HMI
        GVL_HMI.HMIAnimation.sLoadTextRecovery := 'Metering Rinse 1';
        iStepCounter := 1;

    1:  // Initialization: wait solenoids at IDLE (safety/flow configuration)
        // fbSolenoidControl could also be used if re-enabled in the future
        // fbSolenoidControl(bExecute := TRUE, eSolenoidSet := E_SolenoidSet.IDLE);

        IF GVL_IO.gSetSolenoidControl.Idle() THEN
            iStepCounter := 2;
        END_IF

    2:  // Set valves for Rinse 1 (position comes from aSolventN[1])
        FOR i := 1 TO 5 DO
            IF NOT bMoveValveDone[i] THEN
                bMoveValveDone[i] := GVL_Motion.aValvesObj[i].MoveValve(
                    iPosition := GVL_Recipe.stActiveRecipe.stSolventsTimes.aSolventN[1],
                    rVelocity := GVL_Motion.aValves[i].rTargetVel,
                    rAcc      := GVL_Motion.aValves[i].rAcceleration,
                    rDec      := GVL_Motion.aValves[i].rDeceleration
                );
            END_IF
        END_FOR

        IF bMoveValveDone[1] AND bMoveValveDone[2] AND bMoveValveDone[3]
           AND bMoveValveDone[4] AND bMoveValveDone[5]
        THEN
            FOR i := 1 TO 5 DO
                bMoveValveDone[i] := FALSE;
            END_FOR
            iStepCounter := 3;
        END_IF

    3:  // Calculate the distance for each pump (Rinse 1 + dead volume)
        fDistance[1]  := F_VolumeToSteps(GVL_Recipe.stActiveRecipe.stVolumes.aT_IC_Volume[1] +
                                         GVL_Motion.aPumps[1].Rotary.rDeadVolume, 1);
										 
        fDistance[2]  := F_VolumeToSteps(GVL_Recipe.stActiveRecipe.stVolumes.aS0_Volume[1] +
                                         GVL_Motion.aPumps[2].Rotary.rDeadVolume, 2);
										 
        fDistance[3]  := F_VolumeToSteps(GVL_Recipe.stActiveRecipe.stVolumes.aS1_Volume[1] +
                                         GVL_Motion.aPumps[3].Rotary.rDeadVolume, 3);
										 
        fDistance[4]  := F_VolumeToSteps(GVL_Recipe.stActiveRecipe.stVolumes.aS2_Volume[1] +
                                         GVL_Motion.aPumps[4].Rotary.rDeadVolume, 4);
										 
        fDistance[5]  := F_VolumeToSteps(GVL_Recipe.stActiveRecipe.stVolumes.aS3_Volume[1] +
                                         GVL_Motion.aPumps[5].Rotary.rDeadVolume, 5);
										 
        fDistance[6]  := F_VolumeToSteps(GVL_Recipe.stActiveRecipe.stVolumes.aS4_Volume[1] +
                                         GVL_Motion.aPumps[6].Rotary.rDeadVolume, 6);
										 
        fDistance[7]  := F_VolumeToSteps(GVL_Recipe.stActiveRecipe.stVolumes.aS5_Volume[1] +
                                         GVL_Motion.aPumps[7].Rotary.rDeadVolume, 7);
										 
        fDistance[8]  := F_VolumeToSteps(GVL_Recipe.stActiveRecipe.stVolumes.aS6_Volume[1] +
                                         GVL_Motion.aPumps[8].Rotary.rDeadVolume, 8);
										 
        fDistance[9]  := F_VolumeToSteps(GVL_Recipe.stActiveRecipe.stVolumes.aS7_Volume[1] +
                                         GVL_Motion.aPumps[9].Rotary.rDeadVolume, 9);
										 
        fDistance[10] := F_VolumeToSteps(GVL_Recipe.stActiveRecipe.stVolumes.aF_Volume[1] +
                                         GVL_Motion.aPumps[10].Rotary.rDeadVolume, 10);

        iStepCounter := 4;

    4:  // Perform rotary movement for metering (positive movement)
        FOR i := 1 TO 10 DO
            IF NOT bMovePumpDone[i] THEN
                bMovePumpDone[i] := GVL_Motion.aPumpsRotary[i].MoveRelative(
                    Distance := fDistance[i],
                    Velocity := GVL_Settings.stPumpParameters.iMeterVelocity * 6,
                    Acc      := GVL_Settings.stPumpParameters.iMeterVelocity * 6,
                    Dec      := GVL_Settings.stPumpParameters.iMeterVelocity
                );
            END_IF
        END_FOR

        IF bMovePumpDone[1] AND bMovePumpDone[2] AND bMovePumpDone[3] AND bMovePumpDone[4] AND
           bMovePumpDone[5] AND bMovePumpDone[6] AND bMovePumpDone[7] AND bMovePumpDone[8] AND
           bMovePumpDone[9] AND bMovePumpDone[10]
        THEN
            FOR i := 1 TO 10 DO
                bMovePumpDone[i] := FALSE;
            END_FOR
            iStepCounter := 5;
        END_IF

    5:  // Signal completion to Recovery FSM
        bMovementComplete := TRUE;

END_CASE
END_ACTION

ACTION MeteringSolvent2:
// ==========================================================================
// MeteringSolvent2
// --------------------------------------------------------------------------
// Purpose:
//   - Meter Solvent 2 volumes from each Andersen stage into the fluidic path.
//   - Positions valves according to recipe aSolventN[2].
//   - Moves all 10 pumps by distance equivalent to Rinse 2 volumes.
//
// Sequence (iStepCounter):
//   0) Set HMI text.
//   1) Ensure solenoids are in IDLE position.
//   2) Move valves [1..5] to solvent-2 position (recipe-dependent).
//   3) Calculate pump distances (Rinse 2 + dead volume).
//   4) Run all pumps forward at metering velocity.
//   5) Set bMovementComplete TRUE.
// ==========================================================================
CASE iStepCounter OF

    0:  // Initialize action / HMI
        GVL_HMI.HMIAnimation.sLoadTextRecovery := 'Metering Rinse 2';
        iStepCounter := 1;

    1:  // Initialization: wait solenoids at IDLE
        // fbSolenoidControl(bExecute := TRUE, eSolenoidSet := E_SolenoidSet.IDLE);

        IF GVL_IO.gSetSolenoidControl.Idle() THEN
            iStepCounter := 2;
        END_IF

    2:  // Set valves for Rinse 2 (position comes from aSolventN[2])
        FOR i := 1 TO 5 DO
            IF NOT bMoveValveDone[i] THEN
                bMoveValveDone[i] := GVL_Motion.aValvesObj[i].MoveValve(
                    iPosition := GVL_Recipe.stActiveRecipe.stSolventsTimes.aSolventN[2],
                    rVelocity := GVL_Motion.aValves[i].rTargetVel,
                    rAcc      := GVL_Motion.aValves[i].rAcceleration,
                    rDec      := GVL_Motion.aValves[i].rDeceleration
                );
            END_IF
        END_FOR

        IF bMoveValveDone[1] AND bMoveValveDone[2] AND bMoveValveDone[3]
           AND bMoveValveDone[4] AND bMoveValveDone[5]
        THEN
            FOR i := 1 TO 5 DO
                bMoveValveDone[i] := FALSE;
            END_FOR
            iStepCounter := 3;
        END_IF

    3:  // Calculate the distance for each pump (Rinse 2 + dead volume)
        fDistance[1]  := F_VolumeToSteps(GVL_Recipe.stActiveRecipe.stVolumes.aT_IC_Volume[2] +
                                         GVL_Motion.aPumps[1].Rotary.rDeadVolume, 1);
										 
        fDistance[2]  := F_VolumeToSteps(GVL_Recipe.stActiveRecipe.stVolumes.aS0_Volume[2] +
                                         GVL_Motion.aPumps[2].Rotary.rDeadVolume, 2);
										 
        fDistance[3]  := F_VolumeToSteps(GVL_Recipe.stActiveRecipe.stVolumes.aS1_Volume[2] +
                                         GVL_Motion.aPumps[3].Rotary.rDeadVolume, 3);
										 
        fDistance[4]  := F_VolumeToSteps(GVL_Recipe.stActiveRecipe.stVolumes.aS2_Volume[2] +
                                         GVL_Motion.aPumps[4].Rotary.rDeadVolume, 4);
										 
        fDistance[5]  := F_VolumeToSteps(GVL_Recipe.stActiveRecipe.stVolumes.aS3_Volume[2] +
                                         GVL_Motion.aPumps[5].Rotary.rDeadVolume, 5);
										 
        fDistance[6]  := F_VolumeToSteps(GVL_Recipe.stActiveRecipe.stVolumes.aS4_Volume[2] +
                                         GVL_Motion.aPumps[6].Rotary.rDeadVolume, 6);
										 
        fDistance[7]  := F_VolumeToSteps(GVL_Recipe.stActiveRecipe.stVolumes.aS5_Volume[2] +
                                         GVL_Motion.aPumps[7].Rotary.rDeadVolume, 7);
										 
        fDistance[8]  := F_VolumeToSteps(GVL_Recipe.stActiveRecipe.stVolumes.aS6_Volume[2] +
                                         GVL_Motion.aPumps[8].Rotary.rDeadVolume, 8);
										 
        fDistance[9]  := F_VolumeToSteps(GVL_Recipe.stActiveRecipe.stVolumes.aS7_Volume[2] +
                                         GVL_Motion.aPumps[9].Rotary.rDeadVolume, 9);
										 
        fDistance[10] := F_VolumeToSteps(GVL_Recipe.stActiveRecipe.stVolumes.aF_Volume[2] +
                                         GVL_Motion.aPumps[10].Rotary.rDeadVolume, 10);

        iStepCounter := 4;

    4:  // Perform rotary movement for metering (positive movement)
        FOR i := 1 TO 10 DO
            IF NOT bMovePumpDone[i] THEN
                bMovePumpDone[i] := GVL_Motion.aPumpsRotary[i].MoveRelative(
                    Distance := fDistance[i],
                    Velocity := GVL_Settings.stPumpParameters.iMeterVelocity * 6,
                    Acc      := GVL_Settings.stPumpParameters.iMeterVelocity * 6,
                    Dec      := GVL_Settings.stPumpParameters.iMeterVelocity
                );
            END_IF
        END_FOR

        IF bMovePumpDone[1] AND bMovePumpDone[2] AND bMovePumpDone[3] AND bMovePumpDone[4] AND
           bMovePumpDone[5] AND bMovePumpDone[6] AND bMovePumpDone[7] AND bMovePumpDone[8] AND
           bMovePumpDone[9] AND bMovePumpDone[10]
        THEN
            FOR i := 1 TO 10 DO
                bMovePumpDone[i] := FALSE;
            END_FOR
            iStepCounter := 5;
        END_IF

    5:  // Signal completion to Recovery FSM
        bMovementComplete := TRUE;

END_CASE
END_ACTION

ACTION MixSolvent1and2:
// ==========================================================================
// MixSolvent1and2
// --------------------------------------------------------------------------
// Purpose:
//   - Mix Solvent 1 and Solvent 2 by recirculating fluid through the system.
//   - Uses Agitate / Recirculation time from aTime[2] and velocity for solvent 2.
//
// Sequence (iStepCounter):
//   0) Set HMI text.
//   1) Move valves [1..5] to position 5 (Recirculation).
//   2) Compute distance per pump from recirculation time and velocity.
//   3) Run all pumps backward (negative Distance) for mixing.
//   4) Set bMovementComplete TRUE.
// ==========================================================================
CASE iStepCounter OF

    0:  // Initialize action / HMI
        GVL_HMI.HMIAnimation.sLoadTextRecovery := 'Mix Solvents 1 and 2';
        iStepCounter := 1;

    1:  // Move valves [1..5] to position 5 (Recirculation)
        FOR i := 1 TO 5 DO
            IF NOT bMoveValveDone[i] THEN
                bMoveValveDone[i] := GVL_Motion.aValvesObj[i].MoveValve(
                    iPosition := 5,
                    rVelocity := GVL_Motion.aValves[i].rTargetVel,
                    rAcc      := GVL_Motion.aValves[i].rAcceleration,
                    rDec      := GVL_Motion.aValves[i].rDeceleration
                );
            END_IF
        END_FOR

        IF bMoveValveDone[1] AND bMoveValveDone[2] AND bMoveValveDone[3]
           AND bMoveValveDone[4] AND bMoveValveDone[5]
        THEN
            FOR i := 1 TO 5 DO
                bMoveValveDone[i] := FALSE;
            END_FOR
            iStepCounter := 2;
        END_IF

    2:  // Calculate rotation distance based on recirculation time (Rinse 2)
        // fRecirculationTime is in seconds (ms → s)
        fRecirculationTime := TO_REAL(TIME_TO_DWORD(GVL_Recipe.stCurrentRecipe.stSolventsTimes.aTime[2]) / 1000);

        FOR i := 1 TO 10 DO
            // Distance = time * speed (converted to steps elsewhere)
            fCalcDistance[i] := fRecirculationTime *
                                (GVL_Recipe.stActiveRecipe.stSolventsTimes.aVelocity[2] * 6);
        END_FOR

        IF fRecirculationTime > 0 THEN
            iStepCounter := 3;
        END_IF

    3:  // Run pumps with calculated distances [negative movement for mixing]
        FOR i := 1 TO 10 DO
            IF NOT bMovePumpDone[i] THEN
                bMovePumpDone[i] := GVL_Motion.aPumpsRotary[i].MoveRelative(
                    Distance := -fCalcDistance[i],
                    Velocity := GVL_Recipe.stActiveRecipe.stSolventsTimes.aVelocity[2] * 6,
                    Acc      := GVL_Recipe.stActiveRecipe.stSolventsTimes.aVelocity[2] * 3,
                    Dec      := GVL_Recipe.stActiveRecipe.stSolventsTimes.aVelocity[2] * 3
                );
            END_IF
        END_FOR

        IF bMovePumpDone[1] AND bMovePumpDone[2] AND bMovePumpDone[3] AND bMovePumpDone[4] AND
           bMovePumpDone[5] AND bMovePumpDone[6] AND bMovePumpDone[7] AND bMovePumpDone[8] AND
           bMovePumpDone[9] AND bMovePumpDone[10]
        THEN
            FOR i := 1 TO 10 DO
                bMovePumpDone[i] := FALSE;
            END_FOR
            iStepCounter := 4;
        END_IF

    4:  // Signal completion to Recovery FSM
        bMovementComplete := TRUE;

END_CASE
END_ACTION

ACTION PrimeNeedles:
// ==========================================================================
// PrimeNeedles
// --------------------------------------------------------------------------
// Purpose:
//   - Prime the needles and final tubing before vial filling.
//   - Moves valves to needles position (6).
//   - Pumps a configured volume (rVialPrimeVol + margin) through needles.
//
// Sequence (iStepCounter):
//   0) Set HMI text.
//   1) Move valves [1..5] to position 6 (Needles).
//   2) Compute pump distances based on rVialPrimeVol (+10µL margin).
//   3) Run pumps backward (negative Distance) to push fluid out of needles.
//   4) Set bMovementComplete TRUE.
// ==========================================================================
CASE iStepCounter OF

    0:  // Initialize action / HMI
        GVL_HMI.HMIAnimation.sLoadTextRecovery := 'Prime Needles';
        iStepCounter := 1;

    1:  // Set valves for needles position (6)
        FOR i := 1 TO 5 DO
            IF NOT bMoveValveDone[i] THEN
                bMoveValveDone[i] := GVL_Motion.aValvesObj[i].MoveValve(
                    iPosition := 6,
                    rVelocity := GVL_Motion.aValves[i].rTargetVel,
                    rAcc      := GVL_Motion.aValves[i].rAcceleration,
                    rDec      := GVL_Motion.aValves[i].rDeceleration
                );
            END_IF
        END_FOR

        IF bMoveValveDone[1] AND bMoveValveDone[2] AND bMoveValveDone[3]
           AND bMoveValveDone[4] AND bMoveValveDone[5]
        THEN
            FOR i := 1 TO 5 DO
                bMoveValveDone[i] := FALSE;
            END_FOR
            iStepCounter := 2;
        END_IF

    2:  // Calculate the distance for each pump (prime volume + margin)
        fDistance[1]  := F_VolumeToSteps(GVL_Recipe.stActiveRecipe.stOtherParams.rVialPrimeVol + 10, 1);
        fDistance[2]  := F_VolumeToSteps(GVL_Recipe.stActiveRecipe.stOtherParams.rVialPrimeVol + 10, 2);
        fDistance[3]  := F_VolumeToSteps(GVL_Recipe.stActiveRecipe.stOtherParams.rVialPrimeVol + 10, 3);
        fDistance[4]  := F_VolumeToSteps(GVL_Recipe.stActiveRecipe.stOtherParams.rVialPrimeVol + 10, 4);
        fDistance[5]  := F_VolumeToSteps(GVL_Recipe.stActiveRecipe.stOtherParams.rVialPrimeVol + 10, 5);
        fDistance[6]  := F_VolumeToSteps(GVL_Recipe.stActiveRecipe.stOtherParams.rVialPrimeVol + 10, 6);
        fDistance[7]  := F_VolumeToSteps(GVL_Recipe.stActiveRecipe.stOtherParams.rVialPrimeVol + 10, 7);
        fDistance[8]  := F_VolumeToSteps(GVL_Recipe.stActiveRecipe.stOtherParams.rVialPrimeVol + 10, 8);
        fDistance[9]  := F_VolumeToSteps(GVL_Recipe.stActiveRecipe.stOtherParams.rVialPrimeVol + 10, 9);
        fDistance[10] := F_VolumeToSteps(GVL_Recipe.stActiveRecipe.stOtherParams.rVialPrimeVol + 10, 10);

        iStepCounter := 3;

    3:  // Perform rotary movement for priming [negative → pumping out]
        FOR i := 1 TO 10 DO
            IF NOT bMovePumpDone[i] THEN
                bMovePumpDone[i] := GVL_Motion.aPumpsRotary[i].MoveRelative(
                    Distance := -fDistance[i],
                    Velocity := GVL_Settings.stPumpParameters.iMeterVelocity * 6,
                    Acc      := GVL_Settings.stPumpParameters.iMeterVelocity * 3,
                    Dec      := GVL_Settings.stPumpParameters.iMeterVelocity * 3
                );
            END_IF
        END_FOR

        IF bMovePumpDone[1] AND bMovePumpDone[2] AND bMovePumpDone[3] AND bMovePumpDone[4] AND
           bMovePumpDone[5] AND bMovePumpDone[6] AND bMovePumpDone[7] AND bMovePumpDone[8] AND
           bMovePumpDone[9] AND bMovePumpDone[10]
        THEN
            FOR i := 1 TO 10 DO
                bMovePumpDone[i] := FALSE;
            END_FOR
            iStepCounter := 4;
        END_IF

    4:  // Signal completion to Recovery FSM
        bMovementComplete := TRUE;

END_CASE
END_ACTION

ACTION RecirculateSolvent1:
// ==========================================================================
// RecirculateSolvent1
// --------------------------------------------------------------------------
// Purpose:
//   - Recirculate Solvent 1 through the system for a configured time
//     to help dissolve and transport particles.
//
// Sequence (iStepCounter):
//   0) Set HMI text.
//   1) Move valves [1..5] to position 5 (Recirculation).
//   2) Calculate distance per pump from recirculation time (Rinse 1).
//   3) Run all pumps backward (negative Distance).
//   4) Set bMovementComplete TRUE.
// ==========================================================================
CASE iStepCounter OF

    0:  // Initialize action / HMI
        GVL_HMI.HMIAnimation.sLoadTextRecovery := 'Recirculate Solvent';
        iStepCounter := 1;

    1:  // Move valves [1..5] to position 5 (Recirculation)
        FOR i := 1 TO 5 DO
            IF NOT bMoveValveDone[i] THEN
                bMoveValveDone[i] := GVL_Motion.aValvesObj[i].MoveValve(
                    iPosition := 5,
                    rVelocity := GVL_Motion.aValves[i].rTargetVel,
                    rAcc      := GVL_Motion.aValves[i].rAcceleration,
                    rDec      := GVL_Motion.aValves[i].rDeceleration
                );
            END_IF
        END_FOR

        IF bMoveValveDone[1] AND bMoveValveDone[2] AND bMoveValveDone[3]
           AND bMoveValveDone[4] AND bMoveValveDone[5]
        THEN
            FOR i := 1 TO 5 DO
                bMoveValveDone[i] := FALSE;
            END_FOR
            iStepCounter := 2;
        END_IF

    2:  // Calculate rotation distance based on recirculation time (Rinse 1)
        fRecirculationTime := TO_REAL(TIME_TO_DWORD(GVL_Recipe.stCurrentRecipe.stSolventsTimes.aTime[1]) / 1000);

        FOR i := 1 TO 10 DO
            fCalcDistance[i] := fRecirculationTime *
                                (GVL_Recipe.stActiveRecipe.stSolventsTimes.aVelocity[1] * 6);
        END_FOR

        IF fRecirculationTime >= 0 THEN
            iStepCounter := 3;
        END_IF

    3:  // Run pumps with calculated distances [negative movement]
        FOR i := 1 TO 10 DO
            IF NOT bMovePumpDone[i] THEN
                bMovePumpDone[i] := GVL_Motion.aPumpsRotary[i].MoveRelative(
                    Distance := -fCalcDistance[i],
                    Velocity := GVL_Recipe.stActiveRecipe.stSolventsTimes.aVelocity[1] * 6,
                    Acc      := GVL_Recipe.stActiveRecipe.stSolventsTimes.aVelocity[1] * 3,
                    Dec      := GVL_Recipe.stActiveRecipe.stSolventsTimes.aVelocity[1] * 3
                );
            END_IF
        END_FOR

        IF bMovePumpDone[1] AND bMovePumpDone[2] AND bMovePumpDone[3] AND bMovePumpDone[4] AND
           bMovePumpDone[5] AND bMovePumpDone[6] AND bMovePumpDone[7] AND bMovePumpDone[8] AND
           bMovePumpDone[9] AND bMovePumpDone[10]
        THEN
            FOR i := 1 TO 10 DO
                bMovePumpDone[i] := FALSE;
            END_FOR
            iStepCounter := 4;
        END_IF

    4:  // Signal completion to Recovery FSM
        bMovementComplete := TRUE;

END_CASE
END_ACTION

METHOD Reset : BOOL
VAR_INPUT
END_VAR
//Init Flags
nPumpWithError  := 0;
nErrorID   		:= 0;
iStepCounter 	:= 0;
eRecoveryState := E_RecoveryState.Idle;

//Output flags
bSuccess := FALSE;
bError := FALSE;

// Control flags
bStart := FALSE;
bMovementComplete := FALSE;

//Recirculate Solvent
fAgitationTime    	:= 0.0;
fRecirculationTime  := 0.0;

FOR i := 1 TO 10 DO
	fCalcDistance[i] := 0;
	fDistance[i] := 0;
END_FOR

//Solvent Soak
bTimerStarted   := FALSE;
bSoakTimerDone  := FALSE;

//Agitate Time
tonAgitateTime1(IN := FALSE);
tonAgitateTime2(IN := FALSE);

//Icon progress reset
GVL_HMI.HMIAnimation.eIconStateRecovery := E_IconState.Waiting;
GVL_HMI.HMIAnimation.rLoadBarLeakTest := 0;
GVL_HMI.HMIAnimation.rLoadBarRecovery := 0;

tStartTime := T#0S;
rElapsedTimeSec := 0.0;
rTotalEstimatedTimeSec := 0.0;
bProgressInitDone := FALSE;
GVL_HMI.HMIAnimation.rLoadBarRecovery := 0.0;

IF NOT bSuccess AND NOT bError THEN
	Reset := TRUE;
	RETURN;
ELSE
	Reset := FALSE;
END_IF
END_METHOD

ACTION SolventSoak:
// ==========================================================================
// SolventSoak
// --------------------------------------------------------------------------
// Purpose:
//   - Keep solvent in contact with Andersen stages for a soak time.
//   - Uses TON "timerSoak" with tSoakTime from recipe.
//   - Sets bMovementComplete when soak time is elapsed.
//
// Behavior:
//   - Each call keeps re-evaluating timer until bSoakTimerDone is TRUE.
// ==========================================================================
GVL_HMI.HMIAnimation.sLoadTextRecovery := 'Solvent Soak';

// Start Soak timer
bTimerStarted := TRUE;

// Evaluate timer completion
IF timerSoak.Q THEN
    // Soak time completed, reset internal flags
    bTimerStarted  := FALSE;
    bSoakTimerDone := TRUE;
END_IF

// Run TON with soak time from recipe
timerSoak(
    IN := bTimerStarted,
    PT := GVL_Recipe.stActiveRecipe.stOtherParams.tSoakTime
);

// When soak timer is done, notify FSM
IF bSoakTimerDone THEN
    bMovementComplete := TRUE;
END_IF
END_ACTION

ACTION WasteRemainingSolvent:
// ==========================================================================
// WasteRemainingSolvent
// --------------------------------------------------------------------------
// Purpose:
//   - Direct any remaining solvent to the waste container.
//   - Moves M3 to waste position and M2 down, then pumps a combined
//     volume of solvent 1 + solvent 2 out to waste.
//
// Sequence (iStepCounter):
//   0) Set HMI text.
//   1) Move valves [1..5] to needles position (6).
//   2) Move M3 to waste position and M2 down to waste height.
//   3) Calculate pump distances based on total volume (Rinse 1 + Rinse 2).
//   4) Run pumps backward (negative Distance) at run velocity.
//   5) Move M2 back to home position.
//   6) Set bMovementComplete TRUE.
// ==========================================================================
CASE iStepCounter OF

    0:  // Initialize action / HMI
        GVL_HMI.HMIAnimation.sLoadTextRecovery := 'Waste Solvent';
        iStepCounter := 1;

    1:  // Set valves into position 6 (Needles) for wasting
        FOR i := 1 TO 5 DO
            IF NOT bMoveValveDone[i] THEN
                bMoveValveDone[i] := GVL_Motion.aValvesObj[i].MoveValve(
                    iPosition := 6,
                    rVelocity := GVL_Motion.aValves[i].rTargetVel,
                    rAcc      := GVL_Motion.aValves[i].rAcceleration,
                    rDec      := GVL_Motion.aValves[i].rDeceleration
                );
            END_IF
        END_FOR

        IF bMoveValveDone[1] AND bMoveValveDone[2] AND bMoveValveDone[3]
           AND bMoveValveDone[4] AND bMoveValveDone[5]
        THEN
            FOR i := 1 TO 5 DO
                bMoveValveDone[i] := FALSE;
            END_FOR
            iStepCounter := 2;
        END_IF

    2:  // M3/M2 Motors movement to waste position
        // M3 → home (used here as waste position)
        IF NOT bMoveM3 THEN
            bMoveM3 := GVL_Motion.aMotors[3].MoveAbsolute(
                rPosition := GVL_Settings.stMachineParam.aM3Position[1],
                rVelocity := GVL_Settings.stMachineParam.rM3Velocity,
                rAcc      := GVL_Settings.stMachineParam.rM3Accleration,
                rDec      := GVL_Settings.stMachineParam.rM3Deceleration
            );
        END_IF

        // After M3 is done, move M2 down to waste height
        IF NOT bMoveM2 AND bMoveM3 THEN
            bMoveM2 := GVL_Motion.aMotors[2].MoveAbsolute(
                rPosition := GVL_Settings.stMachineParam.aM2Position[2],
                rVelocity := GVL_Settings.stMachineParam.rM2Velocity,
                rAcc      := GVL_Settings.stMachineParam.rM2Accleration,
                rDec      := GVL_Settings.stMachineParam.rM2Deceleration
            );
        END_IF

        IF bMoveM2 AND bMoveM3 THEN
            bMoveM2 := FALSE;
            bMoveM3 := FALSE;
            iStepCounter := 3;
        END_IF

    3:  // Calculate distances for each pump (Rinse 1 + Rinse 2 + margin)
        fDistance[1]  := F_VolumeToSteps(GVL_Recipe.stActiveRecipe.stVolumes.aT_IC_Volume[1] +
                                         GVL_Recipe.stActiveRecipe.stVolumes.aT_IC_Volume[2] + 10, 1);
										 
        fDistance[2]  := F_VolumeToSteps(GVL_Recipe.stActiveRecipe.stVolumes.aS0_Volume[1] +
                                         GVL_Recipe.stActiveRecipe.stVolumes.aS0_Volume[2] + 10, 2);
										 
        fDistance[3]  := F_VolumeToSteps(GVL_Recipe.stActiveRecipe.stVolumes.aS1_Volume[1] +
                                         GVL_Recipe.stActiveRecipe.stVolumes.aS1_Volume[2] + 10, 3);
										 
        fDistance[4]  := F_VolumeToSteps(GVL_Recipe.stActiveRecipe.stVolumes.aS2_Volume[1] +
                                         GVL_Recipe.stActiveRecipe.stVolumes.aS2_Volume[2] + 10, 4);
										 
        fDistance[5]  := F_VolumeToSteps(GVL_Recipe.stActiveRecipe.stVolumes.aS3_Volume[1] +
                                         GVL_Recipe.stActiveRecipe.stVolumes.aS3_Volume[2] + 10, 5);
										 
        fDistance[6]  := F_VolumeToSteps(GVL_Recipe.stActiveRecipe.stVolumes.aS4_Volume[1] +
                                         GVL_Recipe.stActiveRecipe.stVolumes.aS4_Volume[2] + 10, 6);
										 
        fDistance[7]  := F_VolumeToSteps(GVL_Recipe.stActiveRecipe.stVolumes.aS5_Volume[1] +
                                         GVL_Recipe.stActiveRecipe.stVolumes.aS5_Volume[2] + 10, 7);
										 
        fDistance[8]  := F_VolumeToSteps(GVL_Recipe.stActiveRecipe.stVolumes.aS6_Volume[1] +
                                         GVL_Recipe.stActiveRecipe.stVolumes.aS6_Volume[2] + 10, 8);
										 
        fDistance[9]  := F_VolumeToSteps(GVL_Recipe.stActiveRecipe.stVolumes.aS7_Volume[1] +
                                         GVL_Recipe.stActiveRecipe.stVolumes.aS7_Volume[2] + 10, 9);
										 
        fDistance[10] := F_VolumeToSteps(GVL_Recipe.stActiveRecipe.stVolumes.aF_Volume[1] +
                                         GVL_Recipe.stActiveRecipe.stVolumes.aF_Volume[2] + 10, 10);

        iStepCounter := 4;

    4:  // Start pumps to waste remaining solvent [negative movement]
        FOR i := 1 TO 10 DO
            IF NOT bMovePumpDone[i] THEN
                bMovePumpDone[i] := GVL_Motion.aPumpsRotary[i].MoveRelative(
                    Distance := -fDistance[i],
                    Velocity := GVL_Settings.stPumpParameters.iRunVelocity * 6,
                    Acc      := GVL_Settings.stPumpParameters.iRunVelocity * 3,
                    Dec      := GVL_Settings.stPumpParameters.iRunVelocity * 3
                );
            END_IF
        END_FOR

        IF bMovePumpDone[1] AND bMovePumpDone[2] AND bMovePumpDone[3] AND bMovePumpDone[4] AND
           bMovePumpDone[5] AND bMovePumpDone[6] AND bMovePumpDone[7] AND bMovePumpDone[8] AND
           bMovePumpDone[9] AND bMovePumpDone[10]
        THEN
            FOR i := 1 TO 10 DO
                bMovePumpDone[i] := FALSE;
            END_FOR
            iStepCounter := 5;
        END_IF

    5:  // Reset M2 position back to home
        IF NOT bMoveM2 THEN
            bMoveM2 := GVL_Motion.aMotors[2].MoveAbsolute(
                rPosition := GVL_Settings.stMachineParam.aM2Position[1],
                rVelocity := GVL_Settings.stMachineParam.rM2Velocity,
                rAcc      := GVL_Settings.stMachineParam.rM2Accleration,
                rDec      := GVL_Settings.stMachineParam.rM2Deceleration
            );
        END_IF

        IF bMoveM2 THEN
            bMoveM2 := FALSE;
            iStepCounter := 6;
        END_IF

    6:  // Signal completion to Recovery FSM
        bMovementComplete := TRUE;

END_CASE
END_ACTION

END_FUNCTION_BLOCK

// ---- POUs/2. AutoCycle/Hardware Control/FB_SolenoidControl.TcPOU
FUNCTION_BLOCK FB_SolenoidControl
VAR_INPUT
    bExecute      : BOOL;  			// Activates control of solenoid valves
    eSolenoidSet  : E_SolenoidSet; 	// Enum with valve configuration
END_VAR

VAR_OUTPUT
    bDone         : BOOL;  			// Indicates that the valves have been positioned correctly
END_VAR

VAR
    eState        : (IDLE, SET_VALVES, DONE);
	bExecPrev    : BOOL := FALSE;   // memória da execução anterior p/ borda
    bRisingEdge  : BOOL;            // pulso de 1 ciclo na subida de bExecute
	
END_VAR

CASE eState OF
    IDLE:
        bDone := FALSE; // Reinicia a flag done

        // Transição: Vai para SET_VALVES se bExecute for TRUE
        IF bExecute THEN
            eState := SET_VALVES;
        END_IF;

    SET_VALVES: // Configuração das saídas
        // Seu CASE eSolenoidSet permanece aqui
        CASE eSolenoidSet OF
            E_SolenoidSet.IDLE:
                GVL_IO.gDigOutputs.bSolenoidValveA := FALSE;
                GVL_IO.gDigOutputs.bSolenoidValveB := FALSE;
                GVL_IO.gDigOutputs.bSolenoidValveC := FALSE;
            E_SolenoidSet.LEAKTEST:
                GVL_IO.gDigOutputs.bSolenoidValveA := TRUE;
                GVL_IO.gDigOutputs.bSolenoidValveB := TRUE;
                GVL_IO.gDigOutputs.bSolenoidValveC := FALSE;
            E_SolenoidSet.LEAKTESTMONITORING:
                GVL_IO.gDigOutputs.bSolenoidValveA := TRUE;
                GVL_IO.gDigOutputs.bSolenoidValveB := FALSE;
                GVL_IO.gDigOutputs.bSolenoidValveC := FALSE;
            E_SolenoidSet.AIRDRY:
                GVL_IO.gDigOutputs.bSolenoidValveA := FALSE;
                GVL_IO.gDigOutputs.bSolenoidValveB := FALSE;
                GVL_IO.gDigOutputs.bSolenoidValveC := TRUE;
        END_CASE;
        
        // Transição: Vai imediatamente para DONE após configurar as válvulas
        eState := DONE;
    
    DONE:
        // Seta a flag de conclusão
        bDone := TRUE;
        
        // Transição: Espera o comando bExecute ser desativado
        IF NOT bExecute THEN
            eState := IDLE;
            // O reset de bDone para FALSE ocorre no estado IDLE
        END_IF;
END_CASE;

END_FUNCTION_BLOCK

// ---- POUs/2. AutoCycle/Stages/FB_MeteringSolvent1.TcPOU
FUNCTION_BLOCK FB_MeteringSolvent1
VAR_INPUT
	bExecute    : BOOL; 	// start (rising-edge)
END_VAR
VAR_OUTPUT
	bBusy       : BOOL;  	// Busy when running
    bDone       : BOOL;		// Done flag
    bError      : BOOL;		// Error flag
	iErrorCode  : DINT; 	// Erro custom code
END_VAR
VAR
	iStepCounter       : INT := 0;
    bMoveValveDone     : ARRAY[1..5] OF BOOL;
    bMovePumpDone      : ARRAY[1..10] OF BOOL;
    fDistance          : ARRAY[1..10] OF REAL;
	bAllMoveDone	   : BOOL := FALSE;
    fbTmrValves        : TON; 	// watchdog valves
    fbTmrPumps         : TON; 	// watchdog pumps
    bExecutePrev       : BOOL;	// Saves the previous state
    i                  : USINT;	//loop for index
END_VAR

// 0) Disparo por borda de subida
IF (bExecute AND NOT bExecutePrev) AND NOT bBusy AND NOT bDone THEN
    bBusy := TRUE;
    bError := FALSE; iErrorCode := 0;
    iStepCounter := 0;

    // Limpa arrays e timers
    FOR i := 1 TO 5 DO bMoveValveDone[i] := FALSE; END_FOR
    FOR i := 1 TO 10 DO bMovePumpDone[i] := FALSE; END_FOR
END_IF
bExecutePrev := bExecute;

// 1) Máquina de estados só roda quando ocupado
IF bBusy THEN
    CASE iStepCounter OF
        0: // Banner HMI
            GVL_HMI.HMIAnimation.sLoadTextRecovery := 'Metering Rinse 1';
            iStepCounter := 1;

        1: // Solenoides em IDLE
            IF GVL_IO.gSetSolenoidControl.Idle() THEN
                // start watchdog de válvulas
                fbTmrValves(IN:=TRUE, PT:=T#10S);
                iStepCounter := 2;
            END_IF

        2: // Setar válvulas p/ solvente 1
            FOR i := 1 TO 5 DO
                IF NOT bMoveValveDone[i] THEN
                    bMoveValveDone[i] := GVL_Motion.aValvesObj[i].MoveValve(
                        iPosition := GVL_Recipe.stActiveRecipe.stSolventsTimes.aSolventN[1],
                        rVelocity := GVL_Motion.aValves[i].rTargetVel,
                        rAcc      := GVL_Motion.aValves[i].rAcceleration,
                        rDec      := GVL_Motion.aValves[i].rDeceleration
                    );
                END_IF
            END_FOR

            IF bMoveValveDone[1] AND bMoveValveDone[2] AND bMoveValveDone[3] AND bMoveValveDone[4] AND bMoveValveDone[5] THEN
                fbTmrValves(IN:=FALSE);
                FOR i := 1 TO 5 DO bMoveValveDone[i] := FALSE; END_FOR
                iStepCounter := 3;
            ELSIF fbTmrValves.Q THEN
                bError := TRUE; iErrorCode := 1001; // timeout válvulas
                iStepCounter := 6;
            END_IF

        3: // Distâncias por bomba
            fDistance[1] := F_VolumeToSteps(rVolume := GVL_Recipe.stActiveRecipe.stVolumes.aT_IC_Volume[1] + GVL_Motion.aPumps[1].Rotary.rDeadVolume, iPumpIndex := 1);
			fDistance[2] := F_VolumeToSteps(rVolume := GVL_Recipe.stActiveRecipe.stVolumes.aS0_Volume[1] + GVL_Motion.aPumps[2].Rotary.rDeadVolume, iPumpIndex := 2);
			fDistance[3] := F_VolumeToSteps(rVolume := GVL_Recipe.stActiveRecipe.stVolumes.aS1_Volume[1] + GVL_Motion.aPumps[3].Rotary.rDeadVolume, iPumpIndex := 3);
			fDistance[4] := F_VolumeToSteps(rVolume := GVL_Recipe.stActiveRecipe.stVolumes.aS2_Volume[1] + GVL_Motion.aPumps[4].Rotary.rDeadVolume, iPumpIndex := 4);
			fDistance[5] := F_VolumeToSteps(rVolume := GVL_Recipe.stActiveRecipe.stVolumes.aS3_Volume[1] + GVL_Motion.aPumps[5].Rotary.rDeadVolume, iPumpIndex := 5);
			fDistance[6] := F_VolumeToSteps(rVolume := GVL_Recipe.stActiveRecipe.stVolumes.aS4_Volume[1] + GVL_Motion.aPumps[6].Rotary.rDeadVolume, iPumpIndex := 6);
			fDistance[7] := F_VolumeToSteps(rVolume := GVL_Recipe.stActiveRecipe.stVolumes.aS5_Volume[1] + GVL_Motion.aPumps[7].Rotary.rDeadVolume, iPumpIndex := 7);
			fDistance[8] := F_VolumeToSteps(rVolume := GVL_Recipe.stActiveRecipe.stVolumes.aS6_Volume[1] + GVL_Motion.aPumps[8].Rotary.rDeadVolume, iPumpIndex := 8);
			fDistance[9] := F_VolumeToSteps(rVolume := GVL_Recipe.stActiveRecipe.stVolumes.aS7_Volume[1] + GVL_Motion.aPumps[9].Rotary.rDeadVolume, iPumpIndex := 9);
			fDistance[10] := F_VolumeToSteps(rVolume := GVL_Recipe.stActiveRecipe.stVolumes.aF_Volume[1] + GVL_Motion.aPumps[10].Rotary.rDeadVolume, iPumpIndex := 10);
            fbTmrPumps(IN:=TRUE, PT:=T#30S);
            iStepCounter := 4;

        4: // Movimentos das bombas
            FOR i := 1 TO 10 DO
                IF NOT bMovePumpDone[i] THEN
                    bMovePumpDone[i] := GVL_Motion.aPumpsRotary[i].MoveRelative(
                        Distance := fDistance[i],
                        Velocity := GVL_Settings.stPumpParameters.iMeterVelocity * 6,
                        Acc      := GVL_SETTINGS.stPumpParameters.iMeterVelocity * 6,
                        Dec      := GVL_SETTINGS.stPumpParameters.iMeterVelocity
                    );
                END_IF
            END_FOR
			
			bAllMoveDone := bMovePumpDone[1] AND bMovePumpDone[2] AND bMovePumpDone[3] AND bMovePumpDone[4] AND 
						   bMovePumpDone[5] AND bMovePumpDone[6] AND bMovePumpDone[7] AND bMovePumpDone[8] AND 
						   bMovePumpDone[9] AND bMovePumpDone[10];
			
            IF bAllMoveDone THEN // helper p/ AND dos 10 itens
                fbTmrPumps(IN:=FALSE);
                FOR i := 1 TO 10 DO bMovePumpDone[i] := FALSE; END_FOR
                iStepCounter := 5;
            ELSIF fbTmrPumps.Q THEN
                bError := TRUE; iErrorCode := 1002; // timeout bombas
                iStepCounter := 6;
            END_IF

        5: // Done
            bBusy := FALSE;
            bDone := TRUE;
            // NÃO limpar aqui; espere bExecute cair para limpar bDone
            // iStepCounter pode permanecer 5 até o chamador reconhecer

        6: // Error
            bBusy := FALSE;
            // bError TRUE e iErrorCode já setados
            // Aguarde reset do chamador
    END_CASE
END_IF

// 2) Limpeza quando o chamador derruba bExecute (ack)
IF NOT bExecute AND NOT bBusy THEN
    // Libera done (acknowledged) para um próximo ciclo
    bDone := FALSE;
    iStepCounter := 0;
END_IF

METHOD Reset : BOOL
VAR_INPUT
END_VAR
Reset := FALSE;

fbTmrValves(IN := FALSE);
fbTmrPumps(IN := FALSE);

bBusy        := FALSE;
bDone        := FALSE;
bError       := FALSE;
iErrorCode   := 0;
iStepCounter := 0;

FOR i:= 1 TO 10 DO
	bMoveValveDone[i] := FALSE;
	fDistance[i] := 0.0;
END_FOR

FOR i:= 1 TO 5 DO
	bMoveValveDone[i] := FALSE;
END_FOR

bAllMoveDone := FALSE;
bExecutePrev := FALSE;

Reset := TRUE;
RETURN;
END_METHOD

END_FUNCTION_BLOCK

// ---- POUs/Functions/F_VolumeToSteps.TcPOU
FUNCTION F_VolumeToSteps : REAL
VAR_INPUT
	rVolume 	: REAL; // Volume in mL
    iPumpIndex	: INT;  // Pump index 1..10
END_VAR
VAR
END_VAR


F_VolumeToSteps := F_VolumeToSteps_Path(
    					rVolume    := rVolume,
    					iPumpIndex := iPumpIndex,
    					ePath      := E_PumpPath.FillJars
						);

END_FUNCTION

// ---- POUs/Functions/F_VolumeToSteps_Path.TcPOU
FUNCTION F_VolumeToSteps_Path : LREAL
VAR_INPUT
	rVolume    : REAL;       // Requested volume [mL]
    iPumpIndex : UINT;        // Pump index 1..10
    ePath      : E_PumpPath; // Path to apply the correct pump factor
END_VAR
VAR
	rFactor            : REAL;
    rDegreesPerRev     : REAL := 360.0;   // Output expects degrees (1 rev = 360°)
    rEpsilon           : REAL := 1E-6;    // Guard to avoid division by zero
	rRevolutions	   : REAL;
	rRevsPlusHalf	   : REAL;
	iRoundedRevs	   : DINT;
	rFinalDegrees	   : REAL;
END_VAR

// --- Basic input validation ---
IF (iPumpIndex < 1) OR (iPumpIndex > 10) THEN
    // Out of range -> return 0 safely
    F_VolumeToSteps_Path := 0.0;
    RETURN;
END_IF

// --- Select the proper pump factor by path ---
CASE ePath OF
    E_PumpPath.FillJars:
        rFactor := GVL_Motion.aPumps[iPumpIndex].Rotary.rPumpFactorFillJars;
    E_PumpPath.FillCalBox:
        rFactor := GVL_Motion.aPumps[iPumpIndex].Rotary.rPumpFactorFillCalBox;
    E_PumpPath.FromCalBox:
        rFactor := GVL_Motion.aPumps[iPumpIndex].Rotary.rPumpFactorFromCalBox;
ELSE
    // Fallback (defensive): default to FillJars
    rFactor := GVL_Motion.aPumps[iPumpIndex].Rotary.rPumpFactorFillJars;
END_CASE

// --- Guard against invalid/zero factor ---
IF ABS(rFactor) <= rEpsilon THEN
    // Factor not calibrated -> return 0 safely
    F_VolumeToSteps_Path := 0.0;
    RETURN;
END_IF

// 1. Calculate the required number of revolutions (pode ser fracionário)
// Revolutions = Volume [mL] / Factor [mL/rev]
rRevolutions := rVolume / rFactor;

// 2. Implement the rounding logic: TRUNC(x + 0.5)
rRevsPlusHalf := rRevolutions + 0.5;

// 3. Truncate the value to get the nearest integer revolution count.
iRoundedRevs := REAL_TO_DINT(TRUNC(rRevsPlusHalf));

// 4. Convert the integer revolutions back to the angular distance in degrees.
rFinalDegrees := DINT_TO_REAL(iRoundedRevs) * rDegreesPerRev;

// --- Return the final angular distance (in degrees) as LREAL for motion control ---
F_VolumeToSteps_Path := REAL_TO_LREAL(rFinalDegrees);

END_FUNCTION

// ---- POUs/2. AutoCycle/Stages/FB_WashingPhase.TcPOU
(*
    FB_WashingPhase
    ------------------------------------------------------------------------
    Purpose:
      - Orchestrates the full "Washing" macro-phase of the ASRS.
      - Sequences all washing-related steps according to the active recipe:
          1) (Optional) Wash 1:
               - Metering_Wash1
               - Recirculate_Wash1
               - Cleaning_Lines_W1
               - Waste_Wash1
          2) (Optional) Wash 2:
               - Metering_Wash2
               - Recirculate_Wash2
               - Cleaning_Lines_W2
               - Waste_Wash2
          3) Marks washing as Completed when all required steps are done.

      - Updates HMI load bar and washing icon during the entire phase.

    Usage:
      - Call cyclically with bExecute = TRUE while the machine is in
        the Washing Phase state.
      - Internal state machine (eWashingState) progresses through
        each washing step depending on recipe configuration.
      - When eWashingState reaches "Completed", bWashingDone = TRUE.

    Inputs:
      - bExecute : BOOL
          TRUE  → start/continue the washing phase.
          FALSE → keeps FB in Idle (no progression).

    Outputs:
      - bWashingDone  : BOOL
          TRUE when all configured washing steps finish successfully.
      - bWashingError : BOOL
          TRUE if the phase enters Error state
          (currently a reserved hook, not fully used yet).

    Side Effects:
      - Writes to global HMI animation:
          GVL_HMI.HMIAnimation.eIconStateWashing
          GVL_HMI.HMIAnimation.sLoadTextWashing
          GVL_HMI.HMIAnimation.rLoadBarWashing
      - Reads recipe configuration to decide whether Wash 1 and/or Wash 2
        are active:
          GVL_Recipe.stActiveRecipe.stSolventsTimes.aSolventN[3] and [4]
*)

FUNCTION_BLOCK FB_WashingPhase
VAR_INPUT
    bExecute : BOOL;  // TRUE to start/maintain the washing phase
END_VAR

VAR_OUTPUT
    bWashingDone  : BOOL; // Washing finished successfully
    bWashingError : BOOL; // Washing error flag (used in Error state)
END_VAR

VAR
    // -----------------------------
    // Internal Washing FSM state
    // -----------------------------
    bStart        : BOOL := FALSE;                       // Local start latch
    eWashingState : E_WashingState := E_WashingState.Idle; // FSM current state

    // -----------------------------
    // Step / movement coordination
    // -----------------------------
    iStepCounter      : UINT := 0;  // Generic step counter for subroutines
    bMovementComplete : BOOL := FALSE; // TRUE when current washing step is done

    // -----------------------------
    // Motion & flow control flags
    // -----------------------------
    bMoveM2        : BOOL := FALSE;              // Vertical motor M2 movement flag
    bMoveValveDone : ARRAY[1..5] OF BOOL;        // Valve movement completion flags
    bMovePumpDone  : ARRAY[1..10] OF BOOL;       // Pump movement completion flags
    fDistance      : ARRAY[1..10] OF REAL;       // Distance for pump moves (volume-based)

    // -----------------------------
    // Recirculation / agitation parameters
    // -----------------------------
    fAgitationTime     : REAL := 0.0;            // Agitation time from recipe
    fRecirculationTime : REAL := 0.0;            // Recirculation time from recipe
    fCalcDistance      : ARRAY[1..10] OF REAL;   // Pump distances based on time

    i : UINT;                                    // Generic loop index (internal use)

    // -----------------------------
    // HMI progress bar animation
    // -----------------------------
    tStartTime             : TIME := T#0S;  // Stores start time of washing phase
    rElapsedTimeSec        : REAL := 0.0;   // Elapsed time in seconds
    rTotalEstimatedTimeSec : REAL := 0.0;   // Total expected washing time
    bProgressInitDone      : BOOL := FALSE; // TRUE once timing estimation is initialized
END_VAR

// ==========================================================================
// 1) Start latch:
//    - When bExecute becomes TRUE for the first time, latch bStart and
//      put FSM into Idle.
// ==========================================================================
IF NOT bStart THEN
    eWashingState := E_WashingState.Idle;
    bStart        := bExecute;
END_IF

// ==========================================================================
// 2) HMI Progress Bar Animation
//    - Only updates while FSM is running (not Idle/Completed).
//    - Uses external EstimateTotalTime() to scale elapsed time into 0..100%.
// ==========================================================================
IF bProgressInitDone
   AND (eWashingState <> E_WashingState.Idle)
   AND (eWashingState <> E_WashingState.Completed)
THEN
    // Elapsed time in seconds since washing start
    rElapsedTimeSec := TO_REAL(TIME() - tStartTime) / 1000.0;

    // Scale elapsed / estimated total into a percentage
    GVL_HMI.HMIAnimation.rLoadBarWashing :=
        MIN(100.0, rElapsedTimeSec / rTotalEstimatedTimeSec * 100.0);
END_IF

// ==========================================================================
// 3) Washing Phase FSM
// ==========================================================================
CASE eWashingState OF

    // ----------------------------------------------------------------------
    // Idle:
    //  - Reset flags and wait for bStart.
    //  - Initializes HMI and progress timing when phase starts.
    // ----------------------------------------------------------------------
    E_WashingState.Idle:

        // Reset output flags in Idle
        bWashingDone  := FALSE;
        bWashingError := FALSE;

        IF bStart THEN
            // Initialize timing for washing progress bar
            tStartTime             := TIME();
            rTotalEstimatedTimeSec := EstimateTotalTime(); // External estimate
            bProgressInitDone      := TRUE;

            // Configure HMI animation for Washing Phase start
            GVL_HMI.HMIAnimation.eIconStateWashing := E_IconState.InProgress;
            GVL_HMI.HMIAnimation.sLoadTextWashing  := 'Starting';
            GVL_HMI.HMIAnimation.rLoadBarWashing   := 0.0;

            // Decide whether Wash 1 is enabled by recipe:
            // aSolventN[3] > 0 → Wash 1 active
            IF GVL_Recipe.stActiveRecipe.stSolventsTimes.aSolventN[3] > 0 THEN
                eWashingState := E_WashingState.Metering_Wash1;
            ELSE
                // If Wash 1 is not active and neither is Wash 2, the phase can
                // jump directly to Completed. Wash 2 check happens later.
                eWashingState := E_WashingState.Completed;
            END_IF
        END_IF


    // ----------------------------------------------------------------------
    // Metering_Wash1:
    //  - Meters solvent for Wash 1 according to recipe.
    // ----------------------------------------------------------------------
    E_WashingState.Metering_Wash1:

        MeteringWash1();

        IF bMovementComplete THEN
            eWashingState    := E_WashingState.Recirculate_Wash1;
            iStepCounter     := 0;
            bMovementComplete := FALSE;
        END_IF


